// SIMATIC STEP 7 (V5.x) project PLC
// CPU: CPU 315-2 DP
// station: P_ADR_BUS
// station: Hardware
// station: SIMATIC 300(1)
// program: Programma S7(1)

// FB 2: know-how protected block, not included

// FB 3: know-how protected block, not included

// FB 4: know-how protected block, not included

// FB 6: know-how protected block, not included

// FC 1: know-how protected block, not included

FUNCTION FC 2 : VOID
VERSION : 0.1
BEGIN
// (block stored without names or comments; labels and parameter names are numbered)
NETWORK
TITLE =
      TAR1  LD 22;
NETWORK
TITLE =
      LAR1  P#L 2.0;
      L     B#16#10;
      T     LB [AR1,P#0.0];
      L     B#16#2;
      T     LB [AR1,P#1.0];
      L     #PARAM5;
      T     LW [AR1,P#2.0];
      L     #PARAM1;
      T     LW [AR1,P#4.0];
      L     P#DBX 0.0;
      L     #PARAM2;
      SLD   3;
      +D;
      T     LD [AR1,P#6.0];
NETWORK
TITLE =
      LAR1  P#L 12.0;
      L     B#16#10;
      T     LB [AR1,P#0.0];
      L     B#16#2;
      T     LB [AR1,P#1.0];
      L     #PARAM5;
      T     LW [AR1,P#2.0];
      L     #PARAM3;
      T     LW [AR1,P#4.0];
      L     P#DBX 0.0;
      L     #PARAM4;
      SLD   3;
      +D;
      T     LD [AR1,P#6.0];
NETWORK
TITLE =
      CALL  SFC 20 (
           $1                       := P#L 2.0,
           $2                       := P#L 0.0,
           $3                       := P#L 12.0);
NETWORK
TITLE =
      LAR1  LD 22;
END_FUNCTION

// FC 5: know-how protected block, not included

FUNCTION FC 8 : VOID
VERSION : 0.1
BEGIN
// (block stored without names or comments; labels and parameter names are numbered)
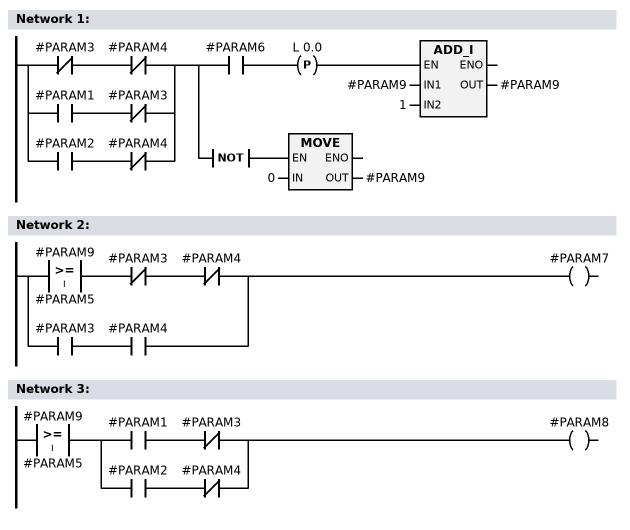
NETWORK
TITLE =
      AN    #PARAM3;
      AN    #PARAM4;
      O;
      A     #PARAM1;
      AN    #PARAM3;
      O;
      A     #PARAM2;
      AN    #PARAM4;
      =     L 1.0;
      A     L 1.0;
      A     #PARAM6;
      FP    L 0.0;
      JNB   M001;
      L     #PARAM9;
      L     1;
      +I;
      T     #PARAM9;
M001: NOP   0;
      A     L 1.0;
      NOT;
      JNB   M002;
      L     0;
      T     #PARAM9;
M002: NOP   0;
NETWORK
TITLE =
      A(;
      L     #PARAM9;
      L     #PARAM5;
      >=I;
      );
      AN    #PARAM3;
      AN    #PARAM4;
      O;
      A     #PARAM3;
      A     #PARAM4;
      =     #PARAM7;
NETWORK
TITLE =
      A(;
      L     #PARAM9;
      L     #PARAM5;
      >=I;
      );
      A(;
      A     #PARAM1;
      AN    #PARAM3;
      O;
      A     #PARAM2;
      AN    #PARAM4;
      );
      =     #PARAM8;
END_FUNCTION

// FC 20: know-how protected block, not included

// FC 21: know-how protected block, not included

// FC 22: know-how protected block, not included

// FC 23: know-how protected block, not included

FUNCTION FC 100 : VOID
VERSION : 0.1
BEGIN
// (block stored without names or comments; labels and parameter names are numbered)
NETWORK
TITLE =
      AN    DB30.DBX 7.0;
      =     DB30.DBX 6.0;
NETWORK
TITLE =
      AN    DB30.DBX 9.0;
      =     DB30.DBX 8.0;
NETWORK
TITLE =
      AN    DB30.DBX 7.1;
      =     DB30.DBX 6.1;
NETWORK
TITLE =
      AN    DB30.DBX 9.1;
      =     DB30.DBX 8.1;
NETWORK
TITLE =
      AN    DB30.DBX 21.1;
      =     DB30.DBX 21.1;
NETWORK
TITLE =
      AN    DB30.DBX 21.2;
      =     DB30.DBX 21.2;
NETWORK
TITLE =
NETWORK
TITLE =
      A     I 6.0;
      =     DB31.DBX 7.7;
NETWORK
TITLE =
      A     I 6.1;
      =     DB31.DBX 107.7;
NETWORK
TITLE =
      A     I 40.5;
      =     DB31.DBX 207.7;
NETWORK
TITLE =
NETWORK
TITLE =
      A     M 10.4;
      A(;
      L     DB30.DBW 34;
      L     18;
      <>I;
      );
      A(;
      L     DB30.DBW 34;
      L     28;
      <>I;
      );
      A(;
      O     I 102.5;
      O     DB30.DBX 509.0;
      );
      =     DB30.DBX 509.0;
NETWORK
TITLE =
      A     M 100.1;
      AN    Q 102.0;
      AN    Q 102.2;
      =     DB30.DBX 509.1;
NETWORK
TITLE =
      A     M 100.3;
      AN    Q 102.1;
      AN    Q 102.3;
      =     DB30.DBX 509.2;
NETWORK
TITLE =
      A     I 60.0;
      A     I 60.1;
      A     I 60.4;
      AN    DB100.DBX 110.0;
      =     DB30.DBX 509.3;
NETWORK
TITLE =
      A     I 60.0;
      A     I 60.1;
      AN    DB100.DBX 110.0;
      =     DB30.DBX 509.4;
NETWORK
TITLE =
      A     I 70.0;
      A     I 70.1;
      A     I 70.4;
      AN    DB100.DBX 110.1;
      =     DB30.DBX 509.5;
NETWORK
TITLE =
      A     I 70.0;
      A     I 70.1;
      AN    DB100.DBX 110.1;
      =     DB30.DBX 509.6;
NETWORK
TITLE =
      A     M 136.2;
      =     DB30.DBX 509.7;
NETWORK
TITLE =
      A     I 80.1;
      AN    DB100.DBX 110.2;
      =     DB30.DBX 511.0;
NETWORK
TITLE =
      A     DB100.DBX 110.6;
      =     DB30.DBX 511.1;
NETWORK
TITLE =
      A     I 90.1;
      AN    DB100.DBX 110.5;
      =     DB30.DBX 511.2;
NETWORK
TITLE =
      A     DB100.DBX 111.0;
      =     DB30.DBX 511.3;
NETWORK
TITLE =
      A     DB100.DBX 111.1;
      =     DB30.DBX 511.4;
NETWORK
TITLE =
      A     M 10.6;
      =     DB30.DBX 511.6;
NETWORK
TITLE =
      A     M 100.0;
      A     M 100.2;
      =     DB30.DBX 511.7;
END_FUNCTION

FUNCTION FC 101 : VOID
VERSION : 0.1
BEGIN
// (block stored without names or comments; labels and parameter names are numbered)
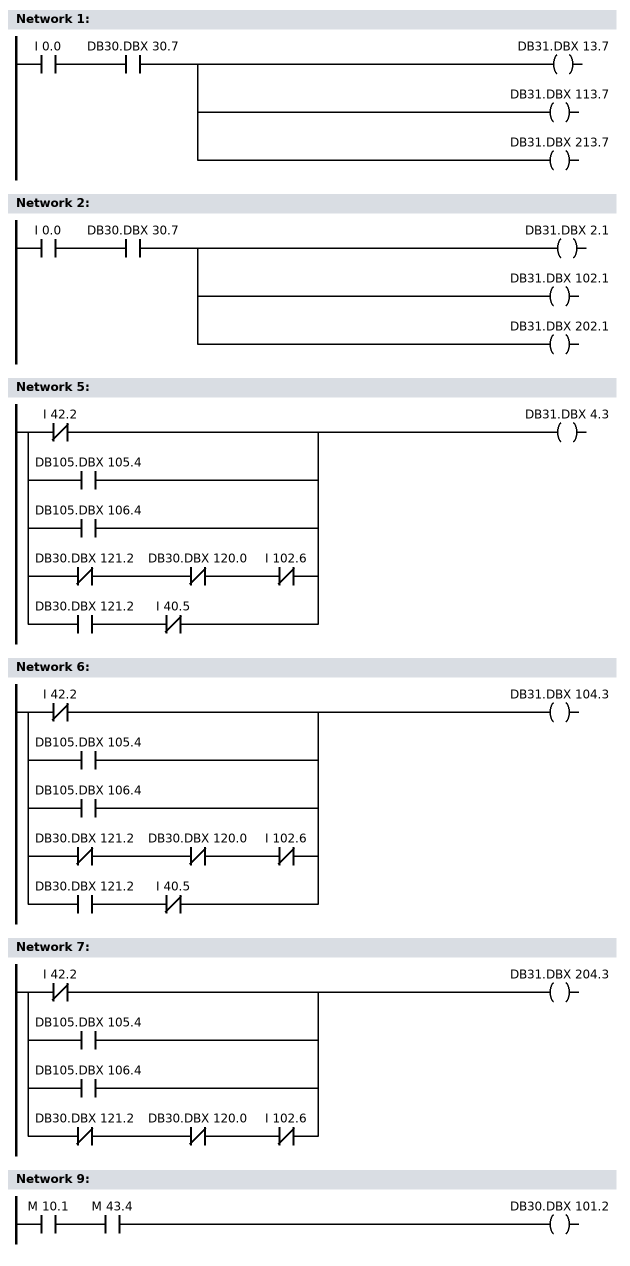
NETWORK
TITLE =
      A     I 0.0;
      A     DB30.DBX 30.7;
      =     DB31.DBX 13.7;
      =     DB31.DBX 113.7;
      =     DB31.DBX 213.7;
NETWORK
TITLE =
      A     I 0.0;
      A     DB30.DBX 30.7;
      =     DB31.DBX 2.1;
      =     DB31.DBX 102.1;
      =     DB31.DBX 202.1;
NETWORK
TITLE =
NETWORK
TITLE =
NETWORK
TITLE =
      ON    I 42.2;
      O     DB105.DBX 105.4;
      O     DB105.DBX 106.4;
      O;
      AN    DB30.DBX 121.2;
      AN    DB30.DBX 120.0;
      AN    I 102.6;
      O;
      A     DB30.DBX 121.2;
      AN    I 40.5;
      =     DB31.DBX 4.3;
NETWORK
TITLE =
      ON    I 42.2;
      O     DB105.DBX 105.4;
      O     DB105.DBX 106.4;
      O;
      AN    DB30.DBX 121.2;
      AN    DB30.DBX 120.0;
      AN    I 102.6;
      O;
      A     DB30.DBX 121.2;
      AN    I 40.5;
      =     DB31.DBX 104.3;
NETWORK
TITLE =
      ON    I 42.2;
      O     DB105.DBX 105.4;
      O     DB105.DBX 106.4;
      O;
      AN    DB30.DBX 121.2;
      AN    DB30.DBX 120.0;
      AN    I 102.6;
      =     DB31.DBX 204.3;
NETWORK
TITLE =
NETWORK
TITLE =
      A     M 10.1;
      A     M 43.4;
      =     DB30.DBX 101.2;
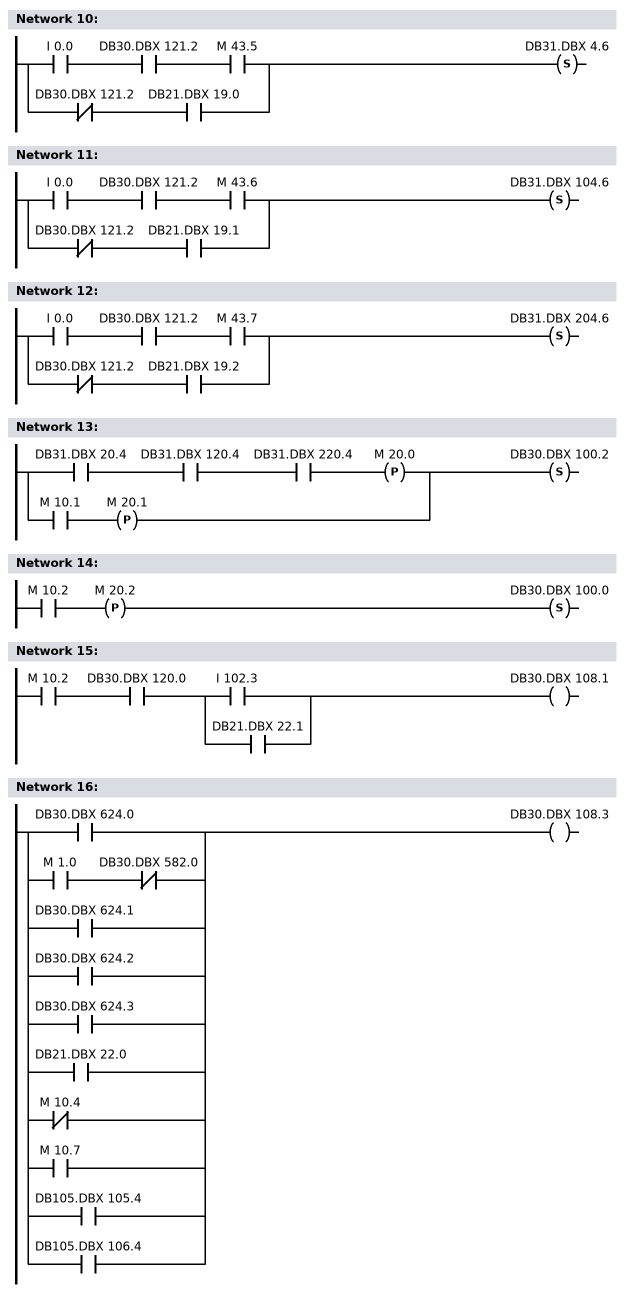
NETWORK
TITLE =
      A     I 0.0;
      A     DB30.DBX 121.2;
      A     M 43.5;
      O;
      AN    DB30.DBX 121.2;
      A     DB21.DBX 19.0;
      S     DB31.DBX 4.6;
NETWORK
TITLE =
      A     I 0.0;
      A     DB30.DBX 121.2;
      A     M 43.6;
      O;
      AN    DB30.DBX 121.2;
      A     DB21.DBX 19.1;
      S     DB31.DBX 104.6;
NETWORK
TITLE =
      A     I 0.0;
      A     DB30.DBX 121.2;
      A     M 43.7;
      O;
      AN    DB30.DBX 121.2;
      A     DB21.DBX 19.2;
      S     DB31.DBX 204.6;
NETWORK
TITLE =
      A     DB31.DBX 20.4;
      A     DB31.DBX 120.4;
      A     DB31.DBX 220.4;
      FP    M 20.0;
      O(;
      A     M 10.1;
      FP    M 20.1;
      );
      S     DB30.DBX 100.2;
NETWORK
TITLE =
      A     M 10.2;
      FP    M 20.2;
      S     DB30.DBX 100.0;
NETWORK
TITLE =
      A     M 10.2;
      A     DB30.DBX 120.0;
      A(;
      O     I 102.3;
      O     DB21.DBX 22.1;
      );
      =     DB30.DBX 108.1;
NETWORK
TITLE =
      O     DB30.DBX 624.0;
      O;
      A     M 1.0;
      AN    DB30.DBX 582.0;
      O     DB30.DBX 624.1;
      O     DB30.DBX 624.2;
      O     DB30.DBX 624.3;
      O     DB21.DBX 22.0;
      ON    M 10.4;
      O     M 10.7;
      O     DB105.DBX 105.4;
      O     DB105.DBX 106.4;
      =     DB30.DBX 108.3;
END_FUNCTION

FUNCTION FC 102 : VOID
VERSION : 0.1
BEGIN
// (block stored without names or comments; labels and parameter names are numbered)
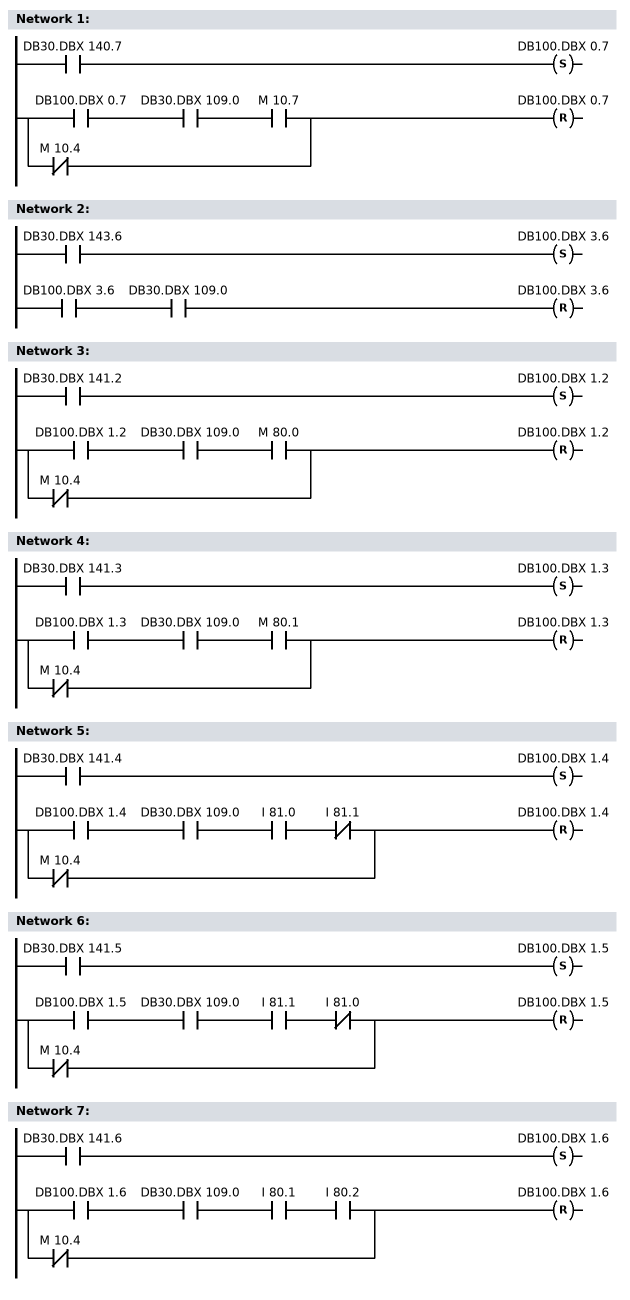
NETWORK
TITLE =
      A     DB30.DBX 140.7;
      S     DB100.DBX 0.7;
      A(;
      A     DB100.DBX 0.7;
      A     DB30.DBX 109.0;
      A     M 10.7;
      ON    M 10.4;
      );
      R     DB100.DBX 0.7;
      NOP   0;
NETWORK
TITLE =
      A     DB30.DBX 143.6;
      S     DB100.DBX 3.6;
      A     DB100.DBX 3.6;
      A     DB30.DBX 109.0;
      R     DB100.DBX 3.6;
      NOP   0;
NETWORK
TITLE =
      A     DB30.DBX 141.2;
      S     DB100.DBX 1.2;
      A(;
      A     DB100.DBX 1.2;
      A     DB30.DBX 109.0;
      A     M 80.0;
      ON    M 10.4;
      );
      R     DB100.DBX 1.2;
      NOP   0;
NETWORK
TITLE =
      A     DB30.DBX 141.3;
      S     DB100.DBX 1.3;
      A(;
      A     DB100.DBX 1.3;
      A     DB30.DBX 109.0;
      A     M 80.1;
      ON    M 10.4;
      );
      R     DB100.DBX 1.3;
      NOP   0;
NETWORK
TITLE =
      A     DB30.DBX 141.4;
      S     DB100.DBX 1.4;
      A(;
      A     DB100.DBX 1.4;
      A     DB30.DBX 109.0;
      A     I 81.0;
      AN    I 81.1;
      ON    M 10.4;
      );
      R     DB100.DBX 1.4;
      NOP   0;
NETWORK
TITLE =
      A     DB30.DBX 141.5;
      S     DB100.DBX 1.5;
      A(;
      A     DB100.DBX 1.5;
      A     DB30.DBX 109.0;
      A     I 81.1;
      AN    I 81.0;
      ON    M 10.4;
      );
      R     DB100.DBX 1.5;
      NOP   0;
NETWORK
TITLE =
      A     DB30.DBX 141.6;
      S     DB100.DBX 1.6;
      A(;
      A     DB100.DBX 1.6;
      A     DB30.DBX 109.0;
      A     I 80.1;
      A     I 80.2;
      ON    M 10.4;
      );
      R     DB100.DBX 1.6;
      NOP   0;
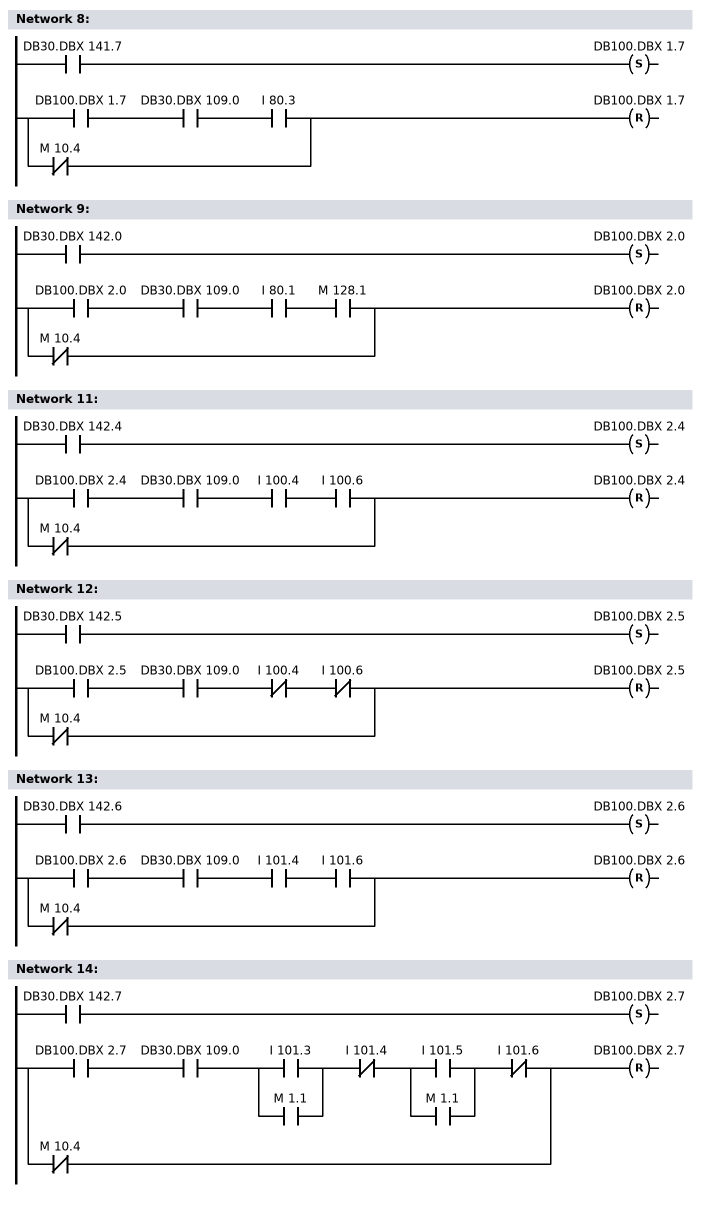
NETWORK
TITLE =
      A     DB30.DBX 141.7;
      S     DB100.DBX 1.7;
      A(;
      A     DB100.DBX 1.7;
      A     DB30.DBX 109.0;
      A     I 80.3;
      ON    M 10.4;
      );
      R     DB100.DBX 1.7;
      NOP   0;
NETWORK
TITLE =
      A     DB30.DBX 142.0;
      S     DB100.DBX 2.0;
      A(;
      A     DB100.DBX 2.0;
      A     DB30.DBX 109.0;
      A     I 80.1;
      A     M 128.1;
      ON    M 10.4;
      );
      R     DB100.DBX 2.0;
      NOP   0;
NETWORK
TITLE =
NETWORK
TITLE =
      A     DB30.DBX 142.4;
      S     DB100.DBX 2.4;
      A(;
      A     DB100.DBX 2.4;
      A     DB30.DBX 109.0;
      A     I 100.4;
      A     I 100.6;
      ON    M 10.4;
      );
      R     DB100.DBX 2.4;
      NOP   0;
NETWORK
TITLE =
      A     DB30.DBX 142.5;
      S     DB100.DBX 2.5;
      A(;
      A     DB100.DBX 2.5;
      A     DB30.DBX 109.0;
      AN    I 100.4;
      AN    I 100.6;
      ON    M 10.4;
      );
      R     DB100.DBX 2.5;
      NOP   0;
NETWORK
TITLE =
      A     DB30.DBX 142.6;
      S     DB100.DBX 2.6;
      A(;
      A     DB100.DBX 2.6;
      A     DB30.DBX 109.0;
      A     I 101.4;
      A     I 101.6;
      ON    M 10.4;
      );
      R     DB100.DBX 2.6;
      NOP   0;
NETWORK
TITLE =
      A     DB30.DBX 142.7;
      S     DB100.DBX 2.7;
      A(;
      A     DB100.DBX 2.7;
      A     DB30.DBX 109.0;
      A(;
      O     I 101.3;
      O     M 1.1;
      );
      AN    I 101.4;
      A(;
      O     I 101.5;
      O     M 1.1;
      );
      AN    I 101.6;
      ON    M 10.4;
      );
      R     DB100.DBX 2.7;
      NOP   0;
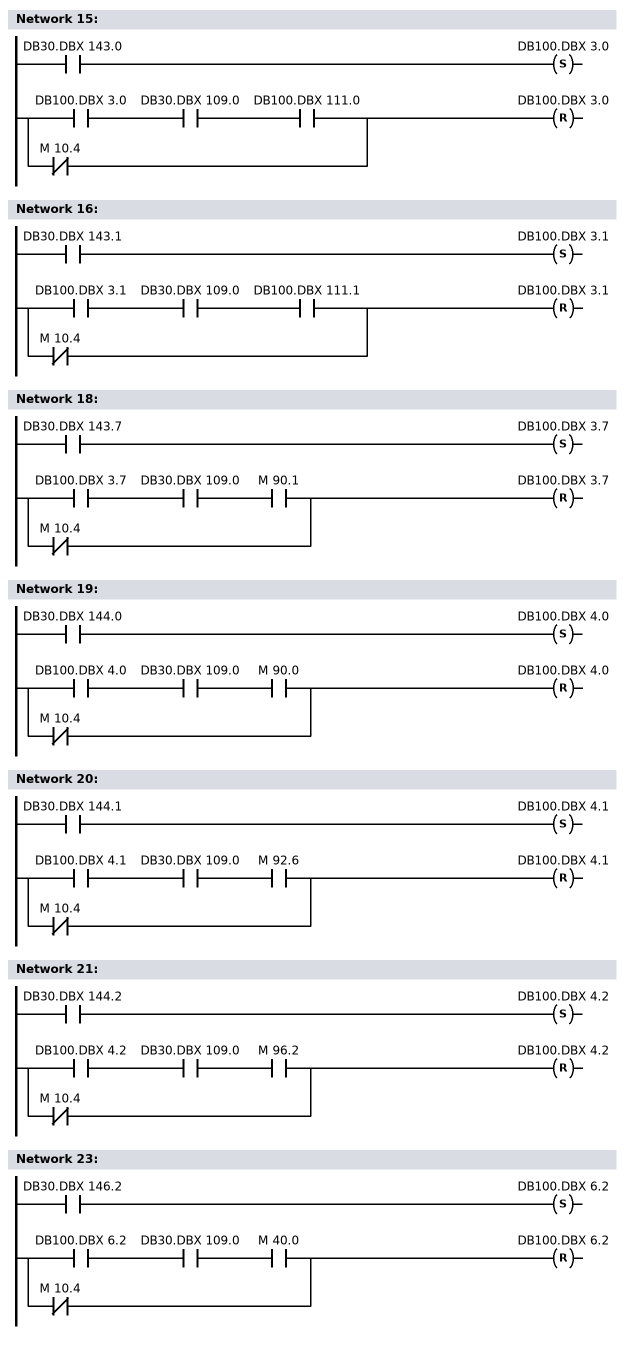
NETWORK
TITLE =
      A     DB30.DBX 143.0;
      S     DB100.DBX 3.0;
      A(;
      A     DB100.DBX 3.0;
      A     DB30.DBX 109.0;
      A     DB100.DBX 111.0;
      ON    M 10.4;
      );
      R     DB100.DBX 3.0;
      NOP   0;
NETWORK
TITLE =
      A     DB30.DBX 143.1;
      S     DB100.DBX 3.1;
      A(;
      A     DB100.DBX 3.1;
      A     DB30.DBX 109.0;
      A     DB100.DBX 111.1;
      ON    M 10.4;
      );
      R     DB100.DBX 3.1;
      NOP   0;
NETWORK
TITLE =
NETWORK
TITLE =
      A     DB30.DBX 143.7;
      S     DB100.DBX 3.7;
      A(;
      A     DB100.DBX 3.7;
      A     DB30.DBX 109.0;
      A     M 90.1;
      ON    M 10.4;
      );
      R     DB100.DBX 3.7;
      NOP   0;
NETWORK
TITLE =
      A     DB30.DBX 144.0;
      S     DB100.DBX 4.0;
      A(;
      A     DB100.DBX 4.0;
      A     DB30.DBX 109.0;
      A     M 90.0;
      ON    M 10.4;
      );
      R     DB100.DBX 4.0;
      NOP   0;
NETWORK
TITLE =
      A     DB30.DBX 144.1;
      S     DB100.DBX 4.1;
      A(;
      A     DB100.DBX 4.1;
      A     DB30.DBX 109.0;
      A     M 92.6;
      ON    M 10.4;
      );
      R     DB100.DBX 4.1;
      NOP   0;
NETWORK
TITLE =
      A     DB30.DBX 144.2;
      S     DB100.DBX 4.2;
      A(;
      A     DB100.DBX 4.2;
      A     DB30.DBX 109.0;
      A     M 96.2;
      ON    M 10.4;
      );
      R     DB100.DBX 4.2;
      NOP   0;
NETWORK
TITLE =
NETWORK
TITLE =
      A     DB30.DBX 146.2;
      S     DB100.DBX 6.2;
      A(;
      A     DB100.DBX 6.2;
      A     DB30.DBX 109.0;
      A     M 40.0;
      ON    M 10.4;
      );
      R     DB100.DBX 6.2;
      NOP   0;
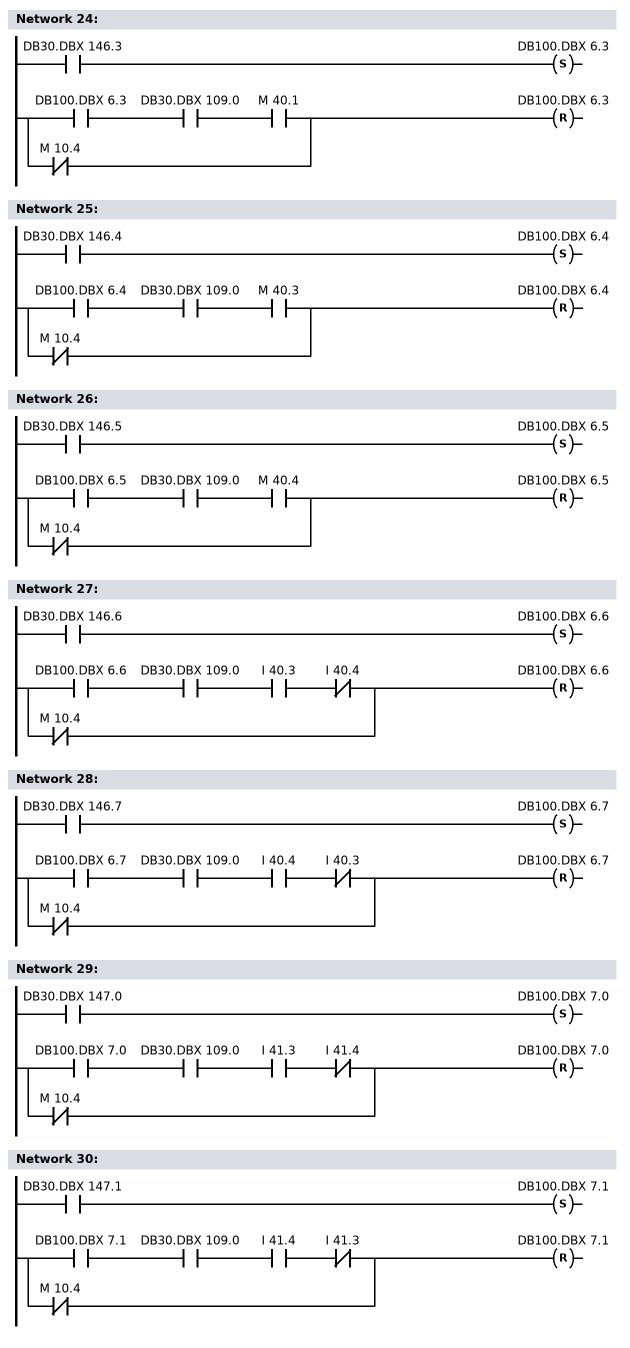
NETWORK
TITLE =
      A     DB30.DBX 146.3;
      S     DB100.DBX 6.3;
      A(;
      A     DB100.DBX 6.3;
      A     DB30.DBX 109.0;
      A     M 40.1;
      ON    M 10.4;
      );
      R     DB100.DBX 6.3;
      NOP   0;
NETWORK
TITLE =
      A     DB30.DBX 146.4;
      S     DB100.DBX 6.4;
      A(;
      A     DB100.DBX 6.4;
      A     DB30.DBX 109.0;
      A     M 40.3;
      ON    M 10.4;
      );
      R     DB100.DBX 6.4;
      NOP   0;
NETWORK
TITLE =
      A     DB30.DBX 146.5;
      S     DB100.DBX 6.5;
      A(;
      A     DB100.DBX 6.5;
      A     DB30.DBX 109.0;
      A     M 40.4;
      ON    M 10.4;
      );
      R     DB100.DBX 6.5;
      NOP   0;
NETWORK
TITLE =
      A     DB30.DBX 146.6;
      S     DB100.DBX 6.6;
      A(;
      A     DB100.DBX 6.6;
      A     DB30.DBX 109.0;
      A     I 40.3;
      AN    I 40.4;
      ON    M 10.4;
      );
      R     DB100.DBX 6.6;
      NOP   0;
NETWORK
TITLE =
      A     DB30.DBX 146.7;
      S     DB100.DBX 6.7;
      A(;
      A     DB100.DBX 6.7;
      A     DB30.DBX 109.0;
      A     I 40.4;
      AN    I 40.3;
      ON    M 10.4;
      );
      R     DB100.DBX 6.7;
      NOP   0;
NETWORK
TITLE =
      A     DB30.DBX 147.0;
      S     DB100.DBX 7.0;
      A(;
      A     DB100.DBX 7.0;
      A     DB30.DBX 109.0;
      A     I 41.3;
      AN    I 41.4;
      ON    M 10.4;
      );
      R     DB100.DBX 7.0;
      NOP   0;
NETWORK
TITLE =
      A     DB30.DBX 147.1;
      S     DB100.DBX 7.1;
      A(;
      A     DB100.DBX 7.1;
      A     DB30.DBX 109.0;
      A     I 41.4;
      AN    I 41.3;
      ON    M 10.4;
      );
      R     DB100.DBX 7.1;
      NOP   0;
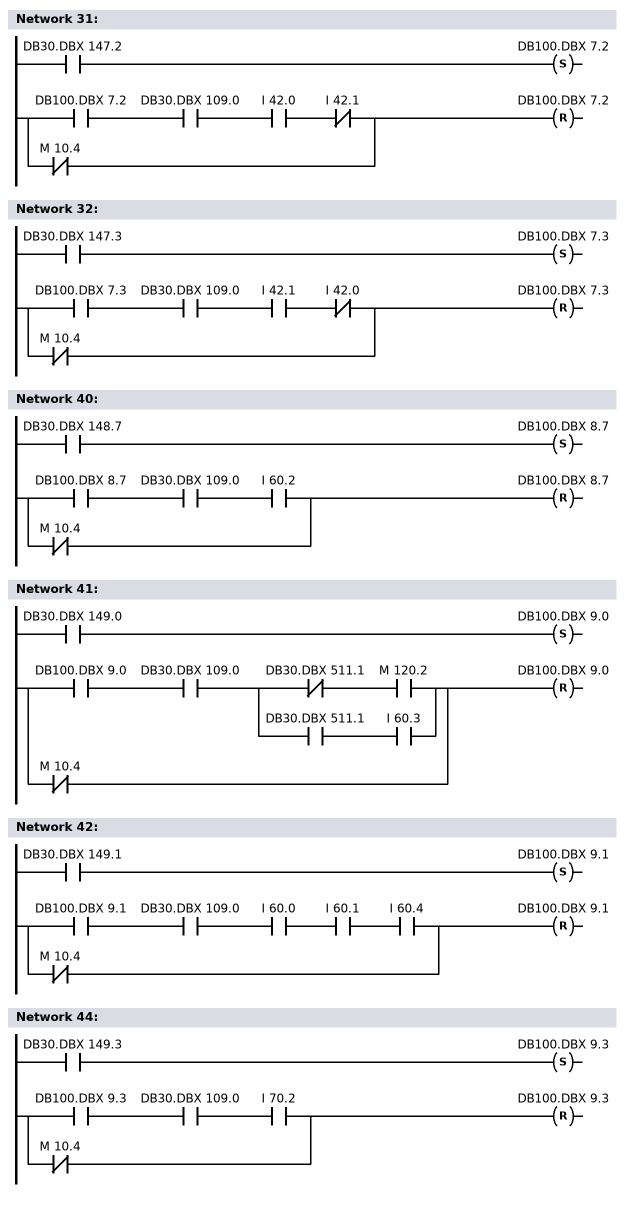
NETWORK
TITLE =
      A     DB30.DBX 147.2;
      S     DB100.DBX 7.2;
      A(;
      A     DB100.DBX 7.2;
      A     DB30.DBX 109.0;
      A     I 42.0;
      AN    I 42.1;
      ON    M 10.4;
      );
      R     DB100.DBX 7.2;
      NOP   0;
NETWORK
TITLE =
      A     DB30.DBX 147.3;
      S     DB100.DBX 7.3;
      A(;
      A     DB100.DBX 7.3;
      A     DB30.DBX 109.0;
      A     I 42.1;
      AN    I 42.0;
      ON    M 10.4;
      );
      R     DB100.DBX 7.3;
      NOP   0;
NETWORK
TITLE =
      A(;
      A     DB30.DBX 147.4;
      S     DB100.DBX 7.4;
      A(;
      A     DB100.DBX 7.4;
      A     DB30.DBX 109.0;
      A     M 132.0;
      ON    M 10.4;
      );
      R     DB100.DBX 7.4;
      A     DB100.DBX 7.4;
      );
      S     M 132.0;
      A     M 132.0;
      AN    DB100.DBX 7.4;
      A     I 40.3;
      AN    I 40.4;
      AN    I 41.3;
      A     I 41.4;
      AN    I 42.0;
      A     I 42.1;
      R     M 132.0;
      NOP   0;
NETWORK
TITLE =
      A(;
      A     DB30.DBX 147.5;
      S     DB100.DBX 7.5;
      A(;
      A     DB100.DBX 7.5;
      A     DB30.DBX 109.0;
      A     M 132.1;
      ON    M 10.4;
      );
      R     DB100.DBX 7.5;
      A     DB100.DBX 7.5;
      );
      S     M 132.1;
      A     M 132.1;
      AN    DB100.DBX 7.5;
      AN    I 40.3;
      A     I 40.4;
      A     I 41.3;
      AN    I 41.4;
      AN    I 42.0;
      A     I 42.1;
      R     M 132.1;
      NOP   0;
NETWORK
TITLE =
      A(;
      A     DB30.DBX 147.6;
      S     DB100.DBX 7.6;
      A(;
      A     DB100.DBX 7.6;
      A     DB30.DBX 109.0;
      A     M 132.2;
      ON    M 10.4;
      );
      R     DB100.DBX 7.6;
      A     DB100.DBX 7.6;
      );
      S     M 132.2;
      A     M 132.2;
      AN    DB100.DBX 7.6;
      A     I 40.3;
      AN    I 40.4;
      AN    I 41.3;
      A     I 41.4;
      A     I 42.0;
      AN    I 42.1;
      R     M 132.2;
      NOP   0;
NETWORK
TITLE =
      A(;
      A     DB30.DBX 147.7;
      S     DB100.DBX 7.7;
      A(;
      A     DB100.DBX 7.7;
      A     DB30.DBX 109.0;
      A     M 132.3;
      ON    M 10.4;
      );
      R     DB100.DBX 7.7;
      A     DB100.DBX 7.7;
      );
      S     M 132.3;
      A     M 132.3;
      AN    DB100.DBX 7.7;
      AN    I 40.3;
      A     I 40.4;
      A     I 41.3;
      AN    I 41.4;
      A     I 42.0;
      AN    I 42.1;
      R     M 132.3;
      NOP   0;
NETWORK
TITLE =
      A(;
      A     DB30.DBX 148.0;
      S     DB100.DBX 8.0;
      A(;
      A     DB100.DBX 8.0;
      A     DB30.DBX 109.0;
      A     M 132.4;
      ON    M 10.4;
      );
      R     DB100.DBX 8.0;
      A     DB100.DBX 8.0;
      );
      S     M 132.4;
      A     M 132.4;
      AN    DB100.DBX 8.0;
      AN    I 40.3;
      A     I 40.4;
      AN    I 41.3;
      A     I 41.4;
      A     I 42.0;
      AN    I 42.1;
      R     M 132.4;
      NOP   0;
NETWORK
TITLE =
      A(;
      A     DB30.DBX 148.1;
      S     DB100.DBX 8.1;
      A(;
      A     DB100.DBX 8.1;
      A     DB30.DBX 109.0;
      A     M 132.5;
      ON    M 10.4;
      );
      R     DB100.DBX 8.1;
      A     DB100.DBX 8.1;
      );
      S     M 132.5;
      A     M 132.5;
      AN    DB100.DBX 8.1;
      AN    I 40.3;
      A     I 40.4;
      AN    I 41.3;
      A     I 41.4;
      AN    I 42.0;
      A     I 42.1;
      R     M 132.5;
      NOP   0;
NETWORK
TITLE =
NETWORK
TITLE =
      A     DB30.DBX 148.7;
      S     DB100.DBX 8.7;
      A(;
      A     DB100.DBX 8.7;
      A     DB30.DBX 109.0;
      A     I 60.2;
      ON    M 10.4;
      );
      R     DB100.DBX 8.7;
      NOP   0;
NETWORK
TITLE =
      A     DB30.DBX 149.0;
      S     DB100.DBX 9.0;
      A(;
      A     DB100.DBX 9.0;
      A     DB30.DBX 109.0;
      A(;
      AN    DB30.DBX 511.1;
      A     M 120.2;
      O;
      A     DB30.DBX 511.1;
      A     I 60.3;
      );
      ON    M 10.4;
      );
      R     DB100.DBX 9.0;
      NOP   0;
NETWORK
TITLE =
      A     DB30.DBX 149.1;
      S     DB100.DBX 9.1;
      A(;
      A     DB100.DBX 9.1;
      A     DB30.DBX 109.0;
      A     I 60.0;
      A     I 60.1;
      A     I 60.4;
      ON    M 10.4;
      );
      R     DB100.DBX 9.1;
      NOP   0;
NETWORK
TITLE =
NETWORK
TITLE =
      A     DB30.DBX 149.3;
      S     DB100.DBX 9.3;
      A(;
      A     DB100.DBX 9.3;
      A     DB30.DBX 109.0;
      A     I 70.2;
      ON    M 10.4;
      );
      R     DB100.DBX 9.3;
      NOP   0;
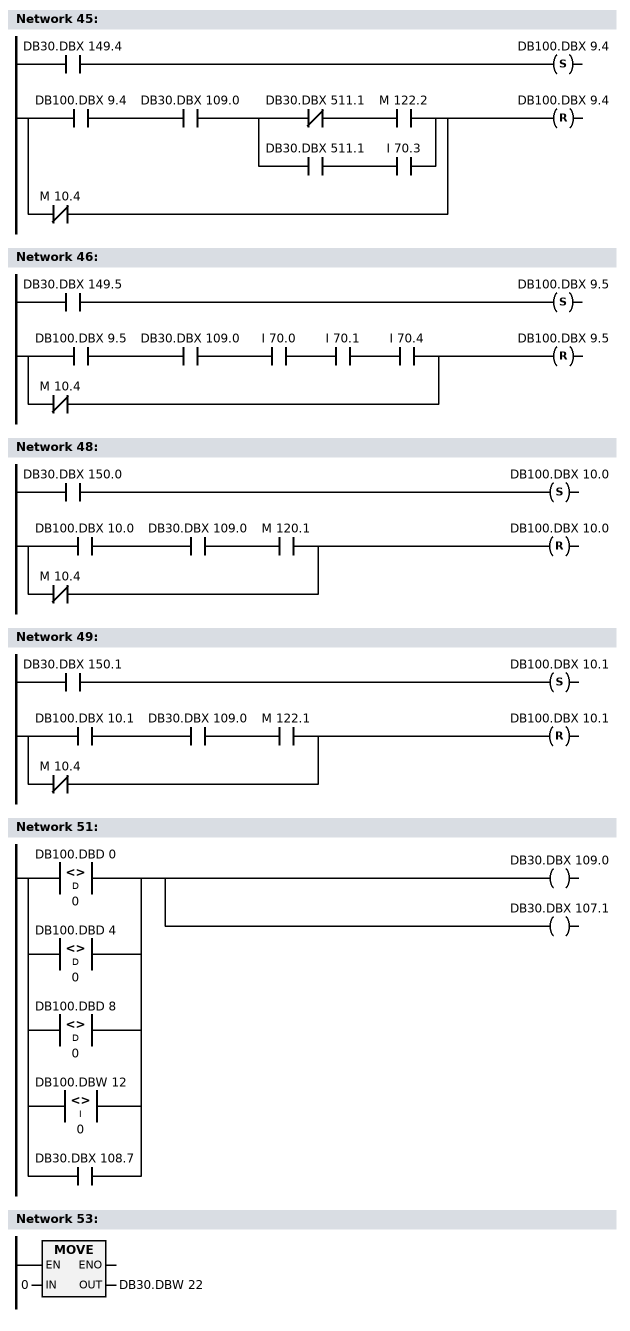
NETWORK
TITLE =
      A     DB30.DBX 149.4;
      S     DB100.DBX 9.4;
      A(;
      A     DB100.DBX 9.4;
      A     DB30.DBX 109.0;
      A(;
      AN    DB30.DBX 511.1;
      A     M 122.2;
      O;
      A     DB30.DBX 511.1;
      A     I 70.3;
      );
      ON    M 10.4;
      );
      R     DB100.DBX 9.4;
      NOP   0;
NETWORK
TITLE =
      A     DB30.DBX 149.5;
      S     DB100.DBX 9.5;
      A(;
      A     DB100.DBX 9.5;
      A     DB30.DBX 109.0;
      A     I 70.0;
      A     I 70.1;
      A     I 70.4;
      ON    M 10.4;
      );
      R     DB100.DBX 9.5;
      NOP   0;
NETWORK
TITLE =
NETWORK
TITLE =
      A     DB30.DBX 150.0;
      S     DB100.DBX 10.0;
      A(;
      A     DB100.DBX 10.0;
      A     DB30.DBX 109.0;
      A     M 120.1;
      ON    M 10.4;
      );
      R     DB100.DBX 10.0;
      NOP   0;
NETWORK
TITLE =
      A     DB30.DBX 150.1;
      S     DB100.DBX 10.1;
      A(;
      A     DB100.DBX 10.1;
      A     DB30.DBX 109.0;
      A     M 122.1;
      ON    M 10.4;
      );
      R     DB100.DBX 10.1;
      NOP   0;
NETWORK
TITLE =
NETWORK
TITLE =
      O(;
      L     DB100.DBD 0;
      L     0;
      <>D;
      );
      O(;
      L     DB100.DBD 4;
      L     0;
      <>D;
      );
      O(;
      L     DB100.DBD 8;
      L     0;
      <>D;
      );
      O(;
      L     DB100.DBW 12;
      L     0;
      <>I;
      );
      O     DB30.DBX 108.7;
      =     DB30.DBX 109.0;
      =     DB30.DBX 107.1;
NETWORK
TITLE =
NETWORK
TITLE =
      L     0;
      T     DB30.DBW 22;
      NOP   0;
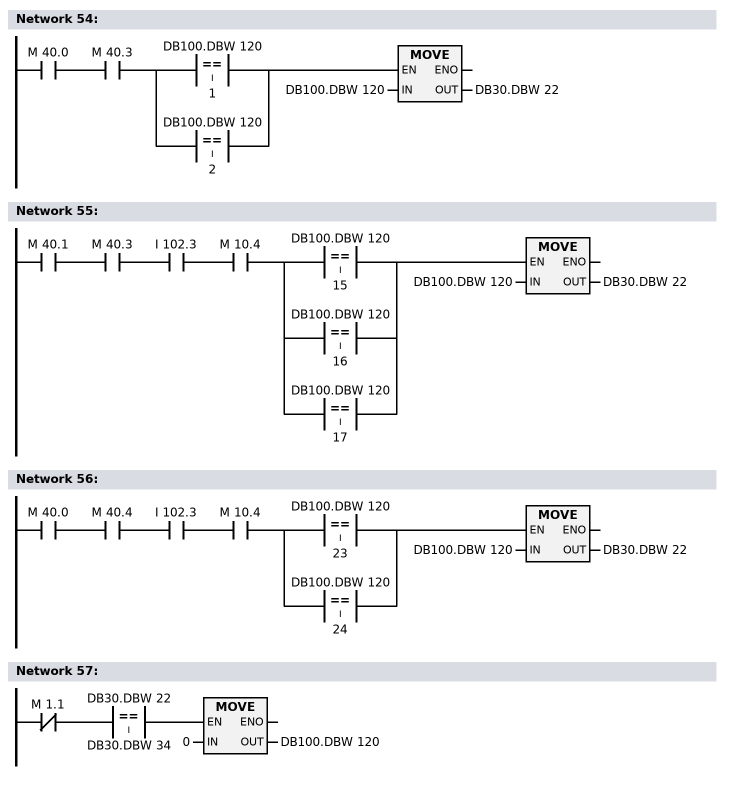
NETWORK
TITLE =
      A     M 40.0;
      A     M 40.3;
      A(;
      O(;
      L     DB100.DBW 120;
      L     1;
      ==I;
      );
      O(;
      L     DB100.DBW 120;
      L     2;
      ==I;
      );
      );
      JNB   M001;
      L     DB100.DBW 120;
      T     DB30.DBW 22;
M001: NOP   0;
NETWORK
TITLE =
      A     M 40.1;
      A     M 40.3;
      A     I 102.3;
      A     M 10.4;
      A(;
      O(;
      L     DB100.DBW 120;
      L     15;
      ==I;
      );
      O(;
      L     DB100.DBW 120;
      L     16;
      ==I;
      );
      O(;
      L     DB100.DBW 120;
      L     17;
      ==I;
      );
      );
      JNB   M002;
      L     DB100.DBW 120;
      T     DB30.DBW 22;
M002: NOP   0;
NETWORK
TITLE =
      A     M 40.0;
      A     M 40.4;
      A     I 102.3;
      A     M 10.4;
      A(;
      O(;
      L     DB100.DBW 120;
      L     23;
      ==I;
      );
      O(;
      L     DB100.DBW 120;
      L     24;
      ==I;
      );
      );
      JNB   M003;
      L     DB100.DBW 120;
      T     DB30.DBW 22;
M003: NOP   0;
NETWORK
TITLE =
      AN    M 1.1;
      A(;
      L     DB30.DBW 22;
      L     DB30.DBW 34;
      ==I;
      );
      JNB   M004;
      L     0;
      T     DB100.DBW 120;
M004: NOP   0;
END_FUNCTION

FUNCTION FC 104 : VOID
AUTHOR : AuD_MCE8
FAMILY : FM357_2
NAME : EXAMPLE5
VERSION : 1.0
BEGIN
// (block stored without names or comments; labels and parameter names are numbered)
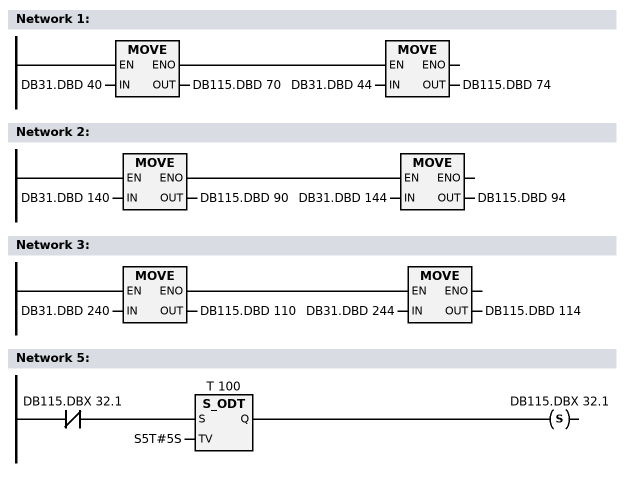
NETWORK
TITLE =
      A(;
      L     DB31.DBD 40;
      T     DB115.DBD 70;
      SET;
      SAVE;
      CLR;
      A     BR;
      );
      JNB   M001;
      L     DB31.DBD 44;
      T     DB115.DBD 74;
M001: NOP   0;
NETWORK
TITLE =
      A(;
      L     DB31.DBD 140;
      T     DB115.DBD 90;
      SET;
      SAVE;
      CLR;
      A     BR;
      );
      JNB   M002;
      L     DB31.DBD 144;
      T     DB115.DBD 94;
M002: NOP   0;
NETWORK
TITLE =
      A(;
      L     DB31.DBD 240;
      T     DB115.DBD 110;
      SET;
      SAVE;
      CLR;
      A     BR;
      );
      JNB   M003;
      L     DB31.DBD 244;
      T     DB115.DBD 114;
M003: NOP   0;
NETWORK
TITLE =
NETWORK
TITLE =
      AN    DB115.DBX 32.1;
      L     S5T#5S;
      SD    T 100;
      NOP   0;
      NOP   0;
      NOP   0;
      A     T 100;
      S     DB115.DBX 32.1;
NETWORK
TITLE =
      A     DB115.DBX 33.3;
      R     DB115.DBX 33.3;
      R     DB115.DBX 32.3;
      JC    M004;
      A     DB115.DBX 32.0;
      FP    DB115.DBX 33.5;
      S     DB115.DBX 32.3;
      O     DB115.DBX 32.7;
      O(;
      A     DB115.DBX 32.5;
      A     DB115.DBX 33.1;
      );
      R     DB115.DBX 32.3;
      R     DB115.DBX 32.0;
M004: CALL  FB 3 , DB 107 (
           DIX 0.0                  := DB115.DBX 32.3,
           DIW 2                    := 3,
           DIW 4                    := W#16#1002,
           DIW 6                    := 10,
           DIW 8                    := 121,
           DID 10                   := P#DBX 30.0,
           DIB 14                   := B#16#1,
           DIW 18                   := 1,
           DIW 132                  := 30,
           DIX 134.0                := DB115.DBX 33.1,
           DIX 134.1                := DB115.DBX 32.7,
           DIW 136                  := LW 0,
           DIW 138                  := W#16#1008,
           DIW 140                  := 1,
           DIW 142                  := 115,
           DID 144                  := P#DBX 0.0);
      L     B#16#0;
      A     DB115.DBX 33.1;
      JCN   M005;
      L     LW 0;
M005: T     DB115.DBW 30;
      A     DB115.DBX 33.2;
      R     DB115.DBX 33.2;
      R     DB115.DBX 32.2;
      JC    M006;
      A     DB115.DBX 32.1;
      FP    DB115.DBX 33.4;
      S     DB115.DBX 32.2;
      A     DB115.DBX 32.6;
      O(;
      A     DB115.DBX 32.4;
      A     DB115.DBX 33.0;
      );
      R     DB115.DBX 32.2;
      R     DB115.DBX 32.1;
M006: CALL  FB 2 , DB 106 (
           DIX 0.0                  := DB115.DBX 32.2,
           DIW 2                    := 8,
           DIW 4                    := W#16#1002,
           DIW 6                    := 10,
           DIW 8                    := 121,
           DID 10                   := P#DBX 30.0,
           DIB 14                   := B#16#1,
           DIW 18                   := 1,
           DIW 20                   := W#16#1002,
           DIW 22                   := 10,
           DIW 24                   := 121,
           DID 26                   := P#DBX 30.0,
           DIB 30                   := B#16#1,
           DIW 34                   := 2,
           DIW 36                   := W#16#1002,
           DIW 38                   := 10,
           DIW 40                   := 121,
           DID 42                   := P#DBX 30.0,
           DIB 46                   := B#16#1,
           DIW 50                   := 3,
           DIW 52                   := W#16#1002,
           DIW 54                   := 10,
           DIW 56                   := 121,
           DID 58                   := P#DBX 30.0,
           DIB 62                   := B#16#1,
           DIW 66                   := 4,
           DIW 68                   := W#16#1002,
           DIW 70                   := 10,
           DIW 72                   := 121,
           DID 74                   := P#DBX 30.0,
           DIB 78                   := B#16#1,
           DIW 82                   := 5,
           DIW 84                   := W#16#1002,
           DIW 86                   := 10,
           DIW 88                   := 121,
           DID 90                   := P#DBX 30.0,
           DIB 94                   := B#16#1,
           DIW 98                   := 6,
           DIW 100                  := W#16#1002,
           DIW 102                  := 10,
           DIW 104                  := 121,
           DID 106                  := P#DBX 30.0,
           DIB 110                  := B#16#1,
           DIW 114                  := 7,
           DIW 116                  := W#16#1002,
           DIW 118                  := 10,
           DIW 120                  := 121,
           DID 122                  := P#DBX 30.0,
           DIB 126                  := B#16#1,
           DIW 130                  := 8,
           DIW 132                  := 30,
           DIX 134.0                := DB115.DBX 33.0,
           DIX 134.1                := DB115.DBX 32.6,
           DIW 136                  := LW 0,
           DIW 138                  := W#16#1008,
           DIW 140                  := 1,
           DIW 142                  := 115,
           DID 144                  := P#DBX 34.0,
           DIW 148                  := W#16#1008,
           DIW 150                  := 1,
           DIW 152                  := 115,
           DID 154                  := P#DBX 38.0,
           DIW 158                  := W#16#1008,
           DIW 160                  := 1,
           DIW 162                  := 115,
           DID 164                  := P#DBX 42.0,
           DIW 168                  := W#16#1008,
           DIW 170                  := 1,
           DIW 172                  := 115,
           DID 174                  := P#DBX 46.0,
           DIW 178                  := W#16#1008,
           DIW 180                  := 1,
           DIW 182                  := 115,
           DID 184                  := P#DBX 50.0,
           DIW 188                  := W#16#1008,
           DIW 190                  := 1,
           DIW 192                  := 115,
           DID 194                  := P#DBX 54.0,
           DIW 198                  := W#16#1008,
           DIW 200                  := 1,
           DIW 202                  := 115,
           DID 204                  := P#DBX 58.0,
           DIW 208                  := W#16#1008,
           DIW 210                  := 1,
           DIW 212                  := 115,
           DID 214                  := P#DBX 62.0);
      L     B#16#0;
      A     DB115.DBX 33.0;
      JCN   M007;
      L     LW 0;
M007: T     DB115.DBW 28;
      BE;
END_FUNCTION

FUNCTION FC 110 : VOID
VERSION : 0.1
BEGIN
// (block stored without names or comments; labels and parameter names are numbered)
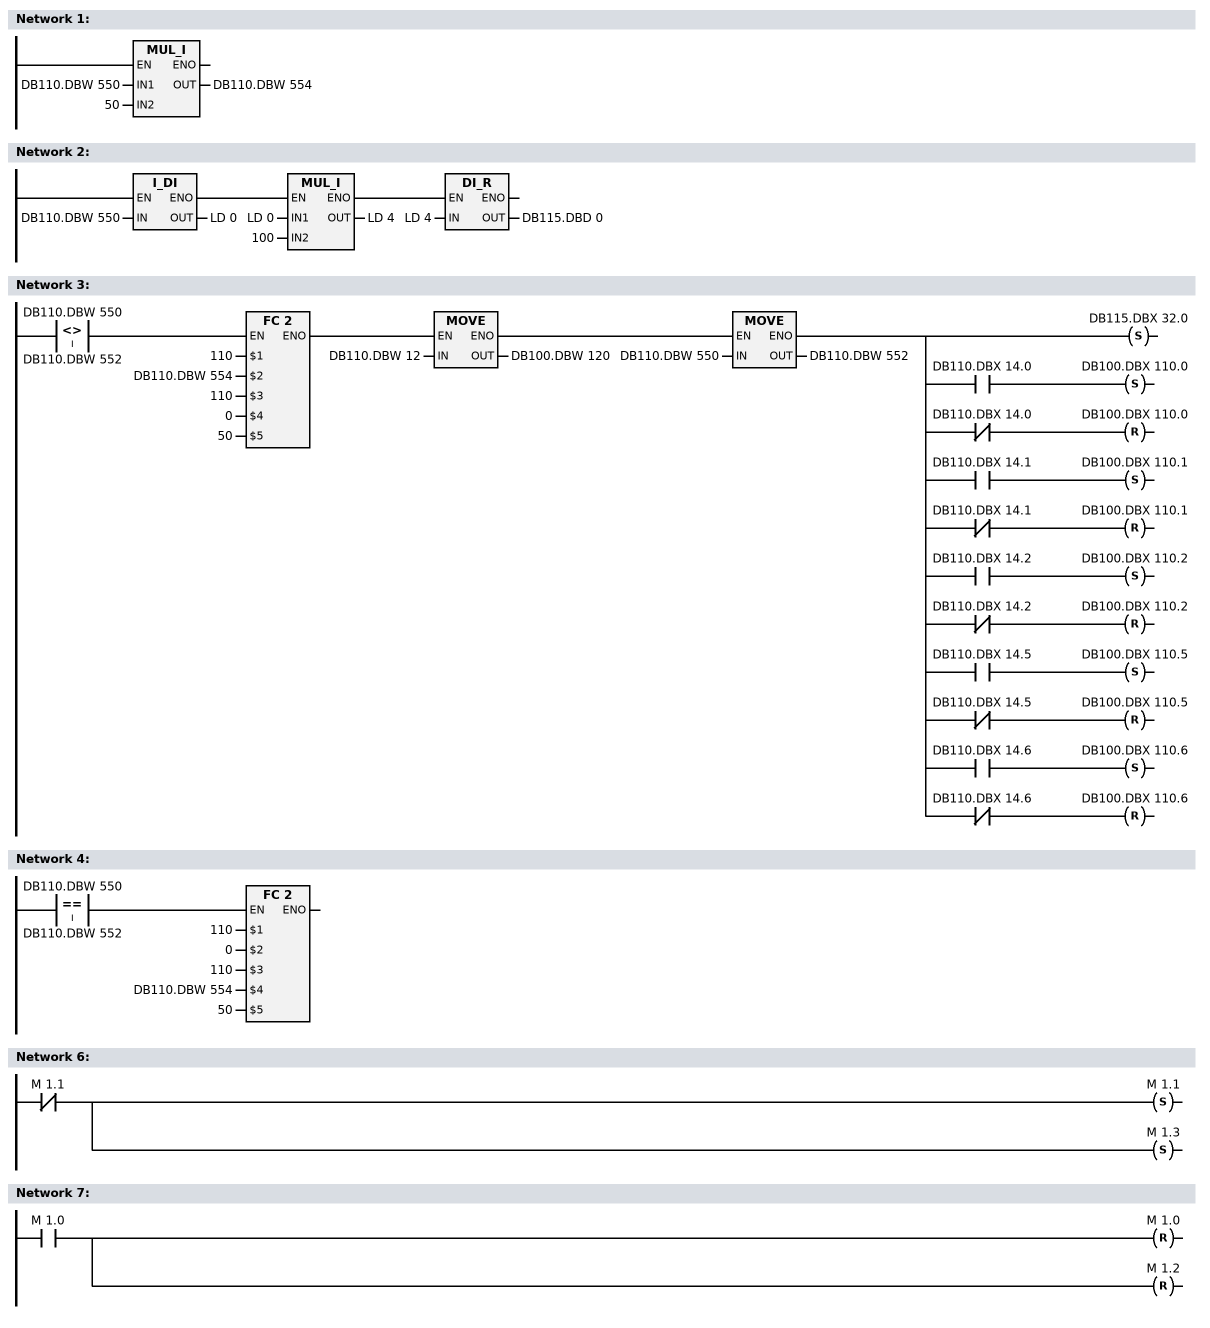
NETWORK
TITLE =
      L     DB110.DBW 550;
      L     50;
      *I;
      T     DB110.DBW 554;
      NOP   0;
NETWORK
TITLE =
      A(;
      A(;
      L     DB110.DBW 550;
      ITD;
      T     LD 0;
      SET;
      SAVE;
      CLR;
      A     BR;
      );
      JNB   M001;
      L     LD 0;
      L     100;
      *I;
      T     LD 4;
      AN    OV;
      SAVE;
      CLR;
M001: A     BR;
      );
      JNB   M002;
      L     LD 4;
      DTR;
      T     DB115.DBD 0;
M002: NOP   0;
NETWORK
TITLE =
      A(;
      A(;
      A(;
      L     DB110.DBW 550;
      L     DB110.DBW 552;
      <>I;
      );
      JNB   M003;
      CALL  FC 2 (
           $1                       := 110,
           $2                       := DB110.DBW 554,
           $3                       := 110,
           $4                       := 0,
           $5                       := 50);
M003: A     BR;
      );
      JNB   M004;
      L     DB110.DBW 12;
      T     DB100.DBW 120;
      SET;
      SAVE;
      CLR;
M004: A     BR;
      );
      JNB   M005;
      L     DB110.DBW 550;
      T     DB110.DBW 552;
      SET;
      SAVE;
      CLR;
M005: A     BR;
      =     L 8.0;
      A     L 8.0;
      BLD   102;
      S     DB115.DBX 32.0;
      A     L 8.0;
      A     DB110.DBX 14.0;
      S     DB100.DBX 110.0;
      A     L 8.0;
      AN    DB110.DBX 14.0;
      R     DB100.DBX 110.0;
      A     L 8.0;
      A     DB110.DBX 14.1;
      S     DB100.DBX 110.1;
      A     L 8.0;
      AN    DB110.DBX 14.1;
      R     DB100.DBX 110.1;
      A     L 8.0;
      A     DB110.DBX 14.2;
      S     DB100.DBX 110.2;
      A     L 8.0;
      AN    DB110.DBX 14.2;
      R     DB100.DBX 110.2;
      A     L 8.0;
      A     DB110.DBX 14.5;
      S     DB100.DBX 110.5;
      A     L 8.0;
      AN    DB110.DBX 14.5;
      R     DB100.DBX 110.5;
      A     L 8.0;
      A     DB110.DBX 14.6;
      S     DB100.DBX 110.6;
      A     L 8.0;
      AN    DB110.DBX 14.6;
      R     DB100.DBX 110.6;
NETWORK
TITLE =
      A(;
      L     DB110.DBW 550;
      L     DB110.DBW 552;
      ==I;
      );
      JNB   M006;
      CALL  FC 2 (
           $1                       := 110,
           $2                       := 0,
           $3                       := 110,
           $4                       := DB110.DBW 554,
           $5                       := 50);
M006: NOP   0;
NETWORK
TITLE =
NETWORK
TITLE =
      AN    M 1.1;
      S     M 1.1;
      S     M 1.3;
NETWORK
TITLE =
      A     M 1.0;
      R     M 1.0;
      R     M 1.2;
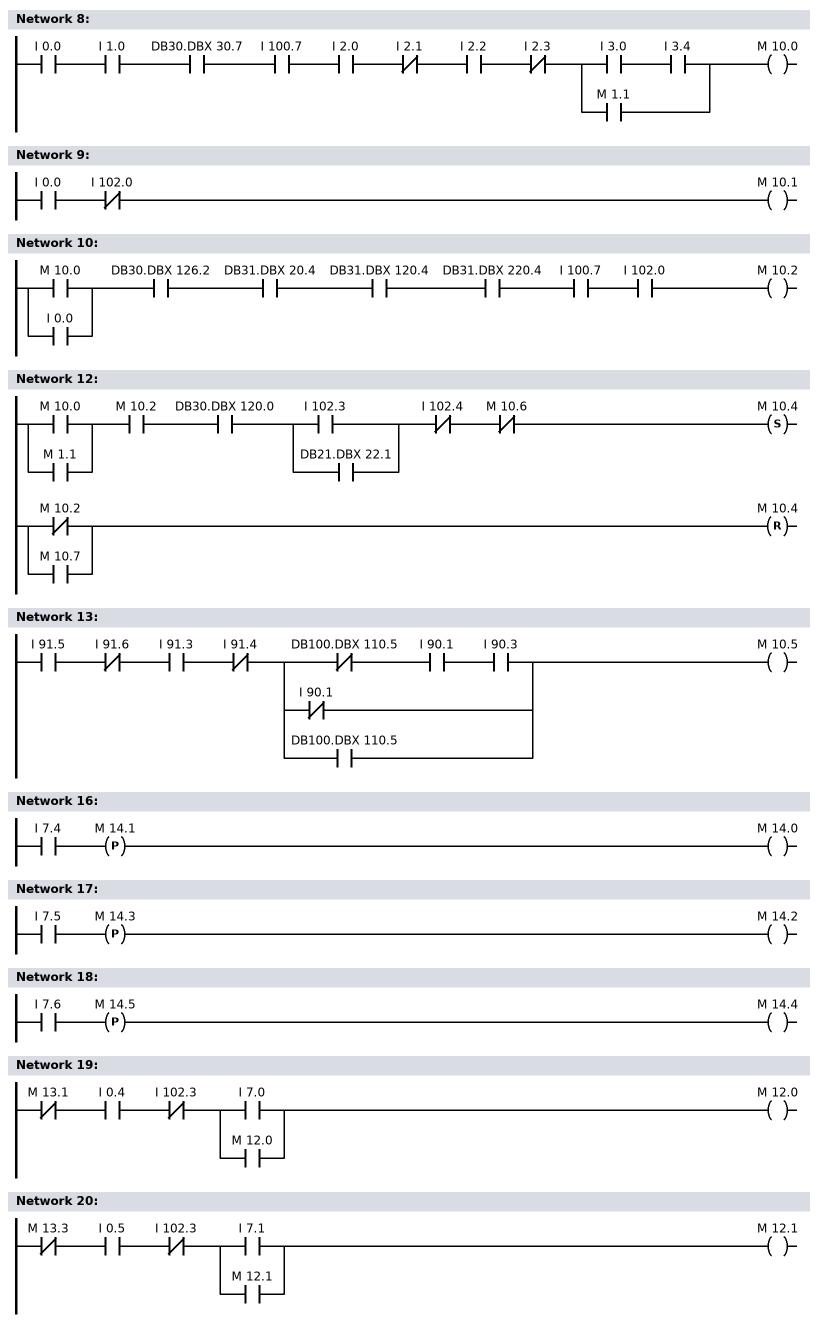
NETWORK
TITLE =
      A     I 0.0;
      A     I 1.0;
      A     DB30.DBX 30.7;
      A     I 100.7;
      A     I 2.0;
      AN    I 2.1;
      A     I 2.2;
      AN    I 2.3;
      A(;
      A     I 3.0;
      A     I 3.4;
      O     M 1.1;
      );
      =     M 10.0;
NETWORK
TITLE =
      A     I 0.0;
      AN    I 102.0;
      =     M 10.1;
NETWORK
TITLE =
      A(;
      O     M 10.0;
      O     I 0.0;
      );
      A     DB30.DBX 126.2;
      A     DB31.DBX 20.4;
      A     DB31.DBX 120.4;
      A     DB31.DBX 220.4;
      A     I 100.7;
      A     I 102.0;
      =     M 10.2;
NETWORK
TITLE =
NETWORK
TITLE =
      A(;
      O     M 10.0;
      O     M 1.1;
      );
      A     M 10.2;
      A     DB30.DBX 120.0;
      A(;
      O     I 102.3;
      O     DB21.DBX 22.1;
      );
      AN    I 102.4;
      AN    M 10.6;
      S     M 10.4;
      A(;
      ON    M 10.2;
      O     M 10.7;
      );
      R     M 10.4;
      NOP   0;
NETWORK
TITLE =
      A     I 91.5;
      AN    I 91.6;
      A     I 91.3;
      AN    I 91.4;
      A(;
      AN    DB100.DBX 110.5;
      A     I 90.1;
      A     I 90.3;
      ON    I 90.1;
      O     DB100.DBX 110.5;
      );
      =     M 10.5;
NETWORK
TITLE =
      A(;
      A     M 10.2;
      A(;
      O     I 102.4;
      O     I 7.0;
      O     I 7.1;
      O     I 7.2;
      );
      S     M 10.6;
      A     M 10.6;
      A(;
      ON    M 10.2;
      O     M 10.7;
      );
      R     M 10.6;
      A     M 10.6;
      );
      A     M 10.5;
      A     DB100.DBX 0.7;
      S     M 10.7;
      A     M 10.7;
      A(;
      O     I 102.3;
      O     DB21.DBX 22.1;
      );
      R     M 10.7;
      NOP   0;
NETWORK
TITLE =
NETWORK
TITLE =
      A     I 7.4;
      BLD   100;
      FP    M 14.1;
      =     M 14.0;
NETWORK
TITLE =
      A     I 7.5;
      BLD   100;
      FP    M 14.3;
      =     M 14.2;
NETWORK
TITLE =
      A     I 7.6;
      BLD   100;
      FP    M 14.5;
      =     M 14.4;
NETWORK
TITLE =
      AN    M 13.1;
      A     I 0.4;
      AN    I 102.3;
      A(;
      O     I 7.0;
      O     M 12.0;
      );
      =     M 12.0;
NETWORK
TITLE =
      AN    M 13.3;
      A     I 0.5;
      AN    I 102.3;
      A(;
      O     I 7.1;
      O     M 12.1;
      );
      =     M 12.1;
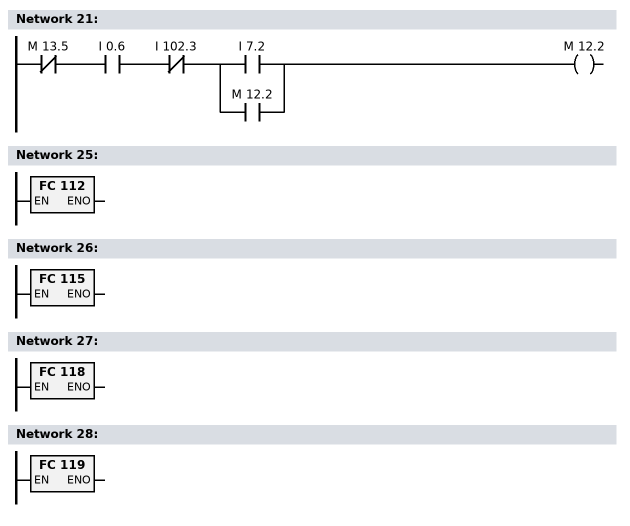
NETWORK
TITLE =
      AN    M 13.5;
      A     I 0.6;
      AN    I 102.3;
      A(;
      O     I 7.2;
      O     M 12.2;
      );
      =     M 12.2;
NETWORK
TITLE =
      A(;
      A(;
      O     M 10.7;
      ON    M 10.4;
      ON    M 10.2;
      );
      AN    Q 3.3;
      A     M 14.0;
      A     M 12.0;
      A(;
      O     M 10.5;
      O     M 1.1;
      );
      AN    M 13.1;
      S     M 13.0;
      A     M 13.0;
      A     M 13.1;
      A     M 14.0;
      A     I 0.4;
      R     M 13.0;
      A     M 13.0;
      );
      S     M 13.1;
      AN    M 13.0;
      A     M 13.1;
      A     M 14.0;
      A     I 0.4;
      R     M 13.1;
      NOP   0;
NETWORK
TITLE =
      A(;
      A(;
      O     M 10.7;
      ON    M 10.4;
      ON    M 10.2;
      );
      AN    Q 3.4;
      A     M 14.2;
      A     M 12.1;
      A(;
      O     M 10.5;
      O     M 1.1;
      );
      AN    M 13.3;
      S     M 13.2;
      A     M 13.2;
      A     M 13.3;
      A     M 14.2;
      A     I 0.5;
      R     M 13.2;
      A     M 13.2;
      );
      S     M 13.3;
      AN    M 13.2;
      A     M 13.3;
      A     M 14.2;
      A     I 0.5;
      R     M 13.3;
      NOP   0;
NETWORK
TITLE =
      A(;
      A(;
      O     M 10.7;
      ON    M 10.4;
      ON    M 10.2;
      );
      AN    Q 3.5;
      A     M 14.4;
      A     M 12.2;
      A(;
      O     M 10.5;
      O     M 1.1;
      );
      AN    M 13.5;
      S     M 13.4;
      A     M 13.4;
      A     M 13.5;
      A     M 14.4;
      A     I 0.6;
      R     M 13.4;
      A     M 13.4;
      );
      S     M 13.5;
      AN    M 13.4;
      A     M 13.5;
      A     M 14.4;
      A     I 0.6;
      R     M 13.5;
      NOP   0;
NETWORK
TITLE =
      CALL  FC 112;
      NOP   0;
NETWORK
TITLE =
      CALL  FC 115;
      NOP   0;
NETWORK
TITLE =
      CALL  FC 118;
      NOP   0;
NETWORK
TITLE =
      CALL  FC 119;
      NOP   0;
END_FUNCTION

FUNCTION FC 112 : VOID
VERSION : 0.1
BEGIN
// (block stored without names or comments; labels and parameter names are numbered)
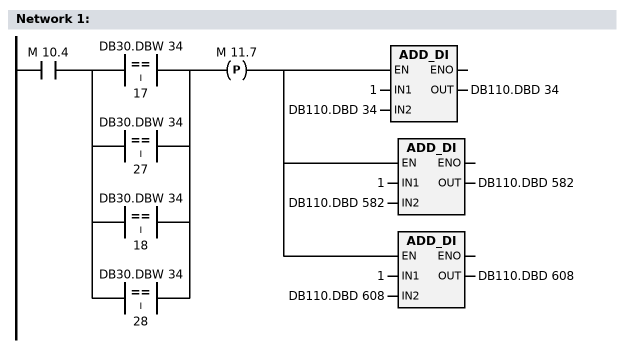
NETWORK
TITLE =
      A     M 10.4;
      A(;
      O(;
      L     DB30.DBW 34;
      L     17;
      ==I;
      );
      O(;
      L     DB30.DBW 34;
      L     27;
      ==I;
      );
      O(;
      L     DB30.DBW 34;
      L     18;
      ==I;
      );
      O(;
      L     DB30.DBW 34;
      L     28;
      ==I;
      );
      );
      FP    M 11.7;
      =     L 0.0;
      A     L 0.0;
      JNB   M001;
      L     1;
      L     DB110.DBD 34;
      +D;
      T     DB110.DBD 34;
M001: NOP   0;
      A     L 0.0;
      JNB   M002;
      L     1;
      L     DB110.DBD 582;
      +D;
      T     DB110.DBD 582;
M002: NOP   0;
      A     L 0.0;
      JNB   M003;
      L     1;
      L     DB110.DBD 608;
      +D;
      T     DB110.DBD 608;
M003: NOP   0;
END_FUNCTION

FUNCTION FC 113 : VOID
VERSION : 0.1
BEGIN
// (block stored without names or comments; labels and parameter names are numbered)
NETWORK
TITLE =
NETWORK
TITLE =
      A(;
      A(;
      A     M 10.4;
      A     M 40.0;
      A     M 40.3;
      A     I 60.0;
      A     I 60.1;
      A(;
      ON    M 120.7;
      O     DB100.DBX 110.1;
      );
      S     M 120.0;
      A(;
      A     M 120.0;
      A     M 120.1;
      ON    M 10.4;
      );
      R     M 120.0;
      A     M 120.0;
      );
      A     DB100.DBX 10.0;
      S     M 120.1;
      A(;
      A     M 120.1;
      A     DB100.DBX 16.1;
      AN    DB100.DBX 10.0;
      ON    M 10.4;
      );
      R     M 120.1;
      A     M 120.1;
      );
      S     DB100.DBX 16.1;
      A     DB100.DBX 16.1;
      A     M 40.3;
      R     DB100.DBX 16.1;
      NOP   0;
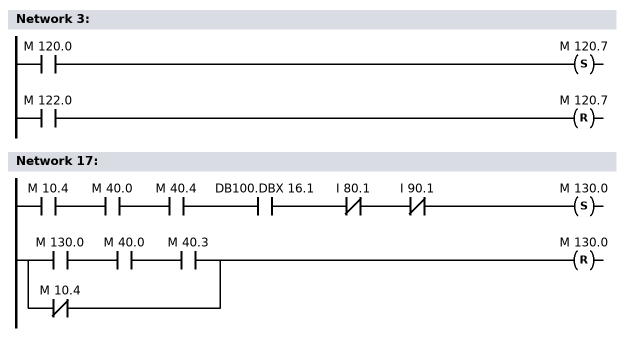
NETWORK
TITLE =
      A     M 120.0;
      S     M 120.7;
      A     M 122.0;
      R     M 120.7;
      NOP   0;
NETWORK
TITLE =
      A(;
      A(;
      A     M 10.4;
      A     M 40.0;
      A     M 40.3;
      AN    I 70.0;
      A     I 70.1;
      A(;
      O     M 120.7;
      O     DB100.DBX 110.0;
      );
      S     M 122.0;
      A(;
      A     M 122.0;
      A     M 122.1;
      ON    M 10.4;
      );
      R     M 122.0;
      A     M 122.0;
      );
      A     DB100.DBX 10.1;
      S     M 122.1;
      A(;
      A     M 122.1;
      A     DB100.DBX 16.1;
      AN    DB100.DBX 10.1;
      ON    M 10.4;
      );
      R     M 122.1;
      A     M 122.1;
      );
      S     DB100.DBX 16.1;
      A     DB100.DBX 16.1;
      A     M 40.3;
      R     DB100.DBX 16.1;
      NOP   0;
NETWORK
TITLE =
NETWORK
TITLE =
      A(;
      A(;
      A     M 10.4;
      A     M 40.0;
      A     M 40.4;
      A     DB100.DBX 16.1;
      A(;
      O     I 80.1;
      O     I 90.1;
      );
      S     M 124.0;
      A(;
      A     M 124.0;
      A     M 124.1;
      ON    M 10.4;
      );
      R     M 124.0;
      A     M 124.0;
      );
      A     DB100.DBX 10.2;
      S     M 124.1;
      A(;
      A     M 124.1;
      A     DB100.DBX 16.5;
      AN    DB100.DBX 10.2;
      ON    M 10.4;
      );
      R     M 124.1;
      A     M 124.1;
      );
      S     DB100.DBX 16.5;
      A     DB100.DBX 16.5;
      A     M 40.3;
      R     DB100.DBX 16.5;
      NOP   0;
NETWORK
TITLE =
NETWORK
TITLE =
      A(;
      A(;
      A     M 10.4;
      A     M 40.1;
      A     M 40.3;
      A(;
      A     DB100.DBX 17.0;
      A(;
      L     DB100.DBW 120;
      L     3;
      ==I;
      );
      O;
      A     DB100.DBX 16.6;
      A(;
      L     DB100.DBW 120;
      L     4;
      ==I;
      );
      );
      S     M 125.0;
      A(;
      A     M 125.0;
      A     M 125.1;
      ON    M 10.4;
      );
      R     M 125.0;
      A     M 125.0;
      );
      A     DB100.DBX 10.3;
      S     M 125.1;
      A(;
      A     M 125.1;
      A     DB100.DBX 16.2;
      AN    DB100.DBX 10.3;
      ON    M 10.4;
      );
      R     M 125.1;
      A     M 125.1;
      );
      A     M 40.1;
      S     DB100.DBX 16.2;
      A     DB100.DBX 16.2;
      A     M 40.0;
      R     DB100.DBX 16.2;
      NOP   0;
NETWORK
TITLE =
      A(;
      A(;
      A     M 10.4;
      A     M 40.0;
      A     M 40.4;
      A(;
      A     DB100.DBX 16.7;
      A(;
      L     DB100.DBW 120;
      L     1;
      ==I;
      );
      O;
      A     DB100.DBX 17.1;
      A(;
      L     DB100.DBW 120;
      L     2;
      ==I;
      );
      );
      S     M 125.2;
      A(;
      A     M 125.0;
      A     M 125.1;
      ON    M 10.4;
      );
      R     M 125.2;
      A     M 125.2;
      );
      A     DB100.DBX 10.3;
      S     M 125.3;
      A(;
      A     M 125.1;
      A     DB100.DBX 16.3;
      AN    DB100.DBX 10.3;
      ON    M 10.4;
      );
      R     M 125.3;
      A     M 125.3;
      );
      A     M 40.4;
      S     DB100.DBX 16.3;
      A     DB100.DBX 16.3;
      A     M 40.3;
      R     DB100.DBX 16.3;
      NOP   0;
NETWORK
TITLE =
NETWORK
TITLE =
      A(;
      A(;
      A     M 10.4;
      A     M 92.6;
      A     M 40.1;
      A     M 40.3;
      A     DB100.DBX 16.6;
      A(;
      L     DB100.DBW 120;
      L     2;
      ==I;
      );
      S     M 126.0;
      A(;
      A     M 126.0;
      A     M 126.1;
      ON    M 10.4;
      );
      R     M 126.0;
      A     M 126.0;
      );
      A     DB100.DBX 10.5;
      S     M 126.1;
      A(;
      A     M 126.1;
      A     DB100.DBX 17.1;
      AN    DB100.DBX 10.5;
      ON    M 10.4;
      );
      R     M 126.1;
      A     M 126.1;
      );
      A     M 40.0;
      A     M 40.4;
      S     DB100.DBX 17.1;
      A     DB100.DBX 17.1;
      A     M 40.3;
      R     DB100.DBX 17.1;
      NOP   0;
NETWORK
TITLE =
      A(;
      A(;
      A     M 10.4;
      A     M 92.6;
      A     M 40.0;
      A     M 40.4;
      A     DB100.DBX 16.5;
      A(;
      O(;
      L     DB100.DBW 120;
      L     1;
      ==I;
      );
      O(;
      L     DB100.DBW 120;
      L     3;
      ==I;
      );
      );
      S     M 126.2;
      A(;
      A     M 126.2;
      A     M 126.3;
      ON    M 10.4;
      );
      R     M 126.2;
      A     M 126.2;
      );
      A     DB100.DBX 10.5;
      S     M 126.3;
      A(;
      A     M 126.3;
      A     DB100.DBX 17.0;
      AN    DB100.DBX 10.5;
      ON    M 10.4;
      );
      R     M 126.3;
      A     M 126.3;
      );
      A     M 40.1;
      A     M 40.3;
      S     DB100.DBX 17.0;
      A     DB100.DBX 17.0;
      A     M 40.0;
      R     DB100.DBX 17.0;
      NOP   0;
NETWORK
TITLE =
NETWORK
TITLE =
      A(;
      A(;
      A     M 10.4;
      A     I 80.0;
      A     I 80.1;
      A     I 80.3;
      A     M 40.1;
      A     M 40.3;
      A     DB100.DBX 17.0;
      A(;
      L     DB100.DBW 120;
      L     1;
      ==I;
      );
      S     M 128.0;
      A(;
      A     M 128.0;
      A     M 128.1;
      ON    M 10.4;
      );
      R     M 128.0;
      A     M 128.0;
      );
      A     DB100.DBX 10.4;
      S     M 128.1;
      A(;
      A     M 128.1;
      A     DB100.DBX 16.7;
      AN    DB100.DBX 10.4;
      ON    M 10.4;
      );
      R     M 128.1;
      A     M 128.1;
      );
      A     M 40.0;
      A     M 40.4;
      S     DB100.DBX 16.7;
      A     DB100.DBX 16.7;
      A     M 40.3;
      R     DB100.DBX 16.7;
      NOP   0;
NETWORK
TITLE =
      A(;
      A(;
      A     M 10.4;
      A     I 80.2;
      A     M 40.0;
      A     M 40.4;
      A     DB100.DBX 16.5;
      A(;
      O(;
      L     DB100.DBW 120;
      L     2;
      ==I;
      );
      O(;
      L     DB100.DBW 120;
      L     4;
      ==I;
      );
      );
      S     M 128.2;
      A(;
      A     M 128.2;
      A     M 128.3;
      ON    M 10.4;
      );
      R     M 128.2;
      A     M 128.2;
      );
      A     DB100.DBX 10.4;
      S     M 128.3;
      A(;
      A     M 128.3;
      A     DB100.DBX 16.6;
      AN    DB100.DBX 10.4;
      ON    M 10.4;
      );
      R     M 128.3;
      A     M 128.3;
      );
      A     M 40.1;
      A     M 40.3;
      S     DB100.DBX 16.6;
      A     DB100.DBX 16.6;
      A     M 40.0;
      R     DB100.DBX 16.6;
      NOP   0;
NETWORK
TITLE =
NETWORK
TITLE =
      A     M 10.4;
      A     M 40.0;
      A     M 40.4;
      A     DB100.DBX 16.1;
      AN    I 80.1;
      AN    I 90.1;
      S     M 130.0;
      A(;
      A     M 130.0;
      A     M 40.0;
      A     M 40.3;
      ON    M 10.4;
      );
      R     M 130.0;
      NOP   0;
END_FUNCTION

FUNCTION FC 115 : VOID
VERSION : 0.1
BEGIN
// (block stored without names or comments; labels and parameter names are numbered)
NETWORK
TITLE =
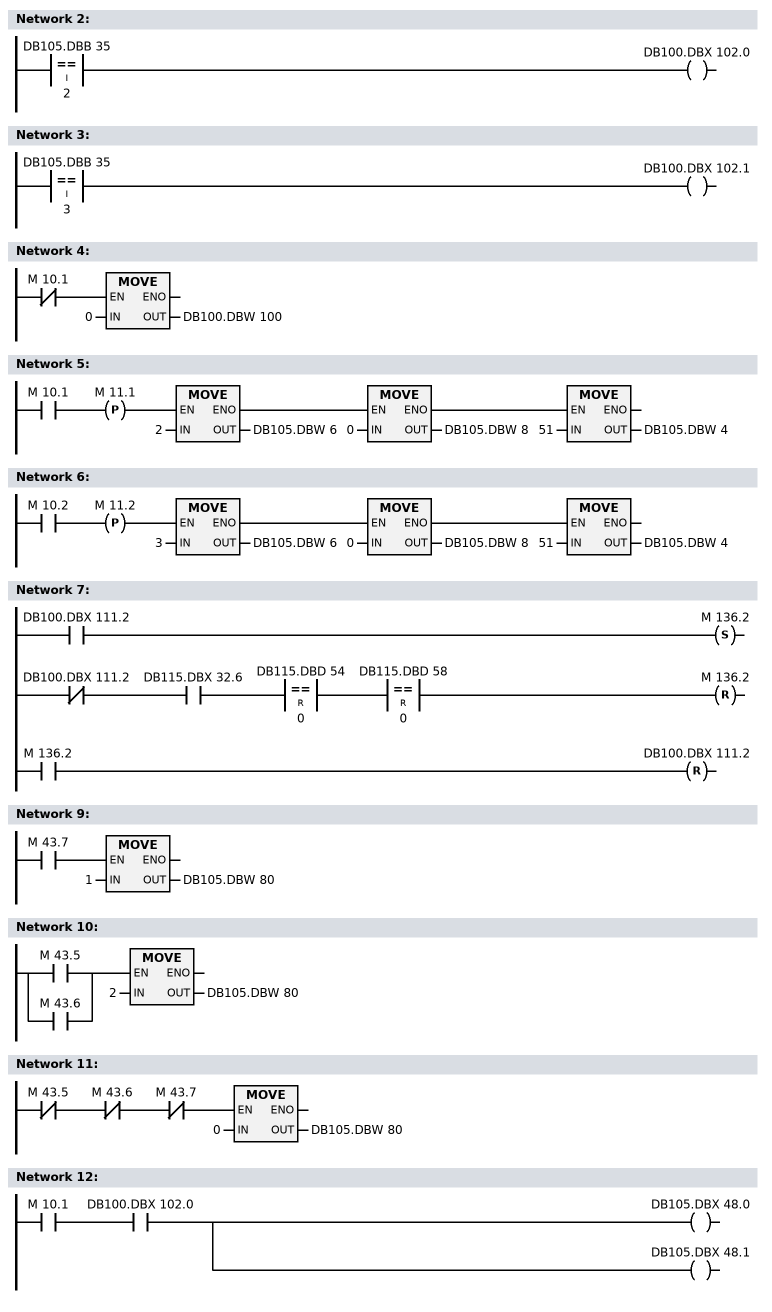
NETWORK
TITLE =
      L     DB105.DBB 35;
      L     2;
      ==I;
      =     DB100.DBX 102.0;
NETWORK
TITLE =
      L     DB105.DBB 35;
      L     3;
      ==I;
      =     DB100.DBX 102.1;
NETWORK
TITLE =
      AN    M 10.1;
      JNB   M001;
      L     0;
      T     DB100.DBW 100;
M001: NOP   0;
NETWORK
TITLE =
      A(;
      A(;
      A     M 10.1;
      FP    M 11.1;
      JNB   M002;
      L     2;
      T     DB105.DBW 6;
      SET;
      SAVE;
      CLR;
M002: A     BR;
      );
      JNB   M003;
      L     0;
      T     DB105.DBW 8;
      SET;
      SAVE;
      CLR;
M003: A     BR;
      );
      JNB   M004;
      L     51;
      T     DB105.DBW 4;
M004: NOP   0;
NETWORK
TITLE =
      A(;
      A(;
      A     M 10.2;
      FP    M 11.2;
      JNB   M005;
      L     3;
      T     DB105.DBW 6;
      SET;
      SAVE;
      CLR;
M005: A     BR;
      );
      JNB   M006;
      L     0;
      T     DB105.DBW 8;
      SET;
      SAVE;
      CLR;
M006: A     BR;
      );
      JNB   M007;
      L     51;
      T     DB105.DBW 4;
M007: NOP   0;
NETWORK
TITLE =
      A     DB100.DBX 111.2;
      S     M 136.2;
      AN    DB100.DBX 111.2;
      A     DB115.DBX 32.6;
      A(;
      L     DB115.DBD 54;
      L     0;
      ==R;
      );
      A(;
      L     DB115.DBD 58;
      L     0;
      ==R;
      );
      R     M 136.2;
      A     M 136.2;
      R     DB100.DBX 111.2;
NETWORK
TITLE =
NETWORK
TITLE =
      A     M 43.7;
      JNB   M008;
      L     1;
      T     DB105.DBW 80;
M008: NOP   0;
NETWORK
TITLE =
      A(;
      O     M 43.5;
      O     M 43.6;
      );
      JNB   M009;
      L     2;
      T     DB105.DBW 80;
M009: NOP   0;
NETWORK
TITLE =
      AN    M 43.5;
      AN    M 43.6;
      AN    M 43.7;
      JNB   M010;
      L     0;
      T     DB105.DBW 80;
M010: NOP   0;
NETWORK
TITLE =
      A     M 10.1;
      A     DB100.DBX 102.0;
      =     DB105.DBX 48.0;
      =     DB105.DBX 48.1;
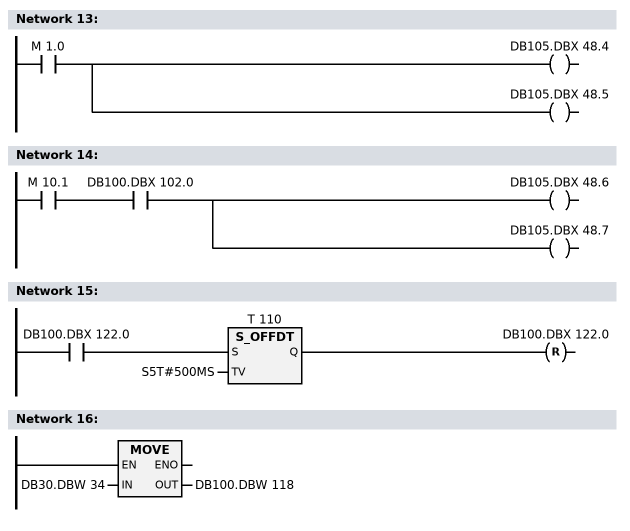
NETWORK
TITLE =
      A     M 1.0;
      =     DB105.DBX 48.4;
      =     DB105.DBX 48.5;
NETWORK
TITLE =
      A     M 10.1;
      A     DB100.DBX 102.0;
      =     DB105.DBX 48.6;
      =     DB105.DBX 48.7;
NETWORK
TITLE =
      A     DB100.DBX 122.0;
      L     S5T#500MS;
      SF    T 110;
      NOP   0;
      NOP   0;
      NOP   0;
      A     T 110;
      R     DB100.DBX 122.0;
NETWORK
TITLE =
      L     DB30.DBW 34;
      T     DB100.DBW 118;
      NOP   0;
END_FUNCTION

FUNCTION FC 118 : VOID
VERSION : 0.1
BEGIN
// (block stored without names or comments; labels and parameter names are numbered)
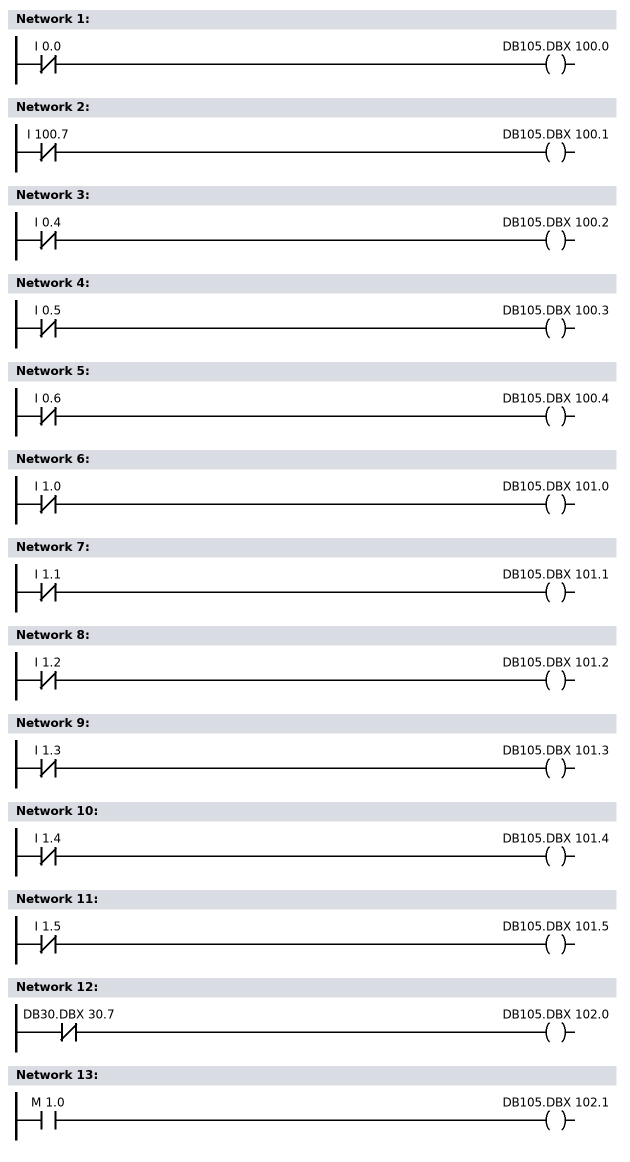
NETWORK
TITLE =
      AN    I 0.0;
      =     DB105.DBX 100.0;
NETWORK
TITLE =
      AN    I 100.7;
      =     DB105.DBX 100.1;
NETWORK
TITLE =
      AN    I 0.4;
      =     DB105.DBX 100.2;
NETWORK
TITLE =
      AN    I 0.5;
      =     DB105.DBX 100.3;
NETWORK
TITLE =
      AN    I 0.6;
      =     DB105.DBX 100.4;
NETWORK
TITLE =
      AN    I 1.0;
      =     DB105.DBX 101.0;
NETWORK
TITLE =
      AN    I 1.1;
      =     DB105.DBX 101.1;
NETWORK
TITLE =
      AN    I 1.2;
      =     DB105.DBX 101.2;
NETWORK
TITLE =
      AN    I 1.3;
      =     DB105.DBX 101.3;
NETWORK
TITLE =
      AN    I 1.4;
      =     DB105.DBX 101.4;
NETWORK
TITLE =
      AN    I 1.5;
      =     DB105.DBX 101.5;
NETWORK
TITLE =
      AN    DB30.DBX 30.7;
      =     DB105.DBX 102.0;
NETWORK
TITLE =
      A     M 1.0;
      =     DB105.DBX 102.1;
NETWORK
TITLE =
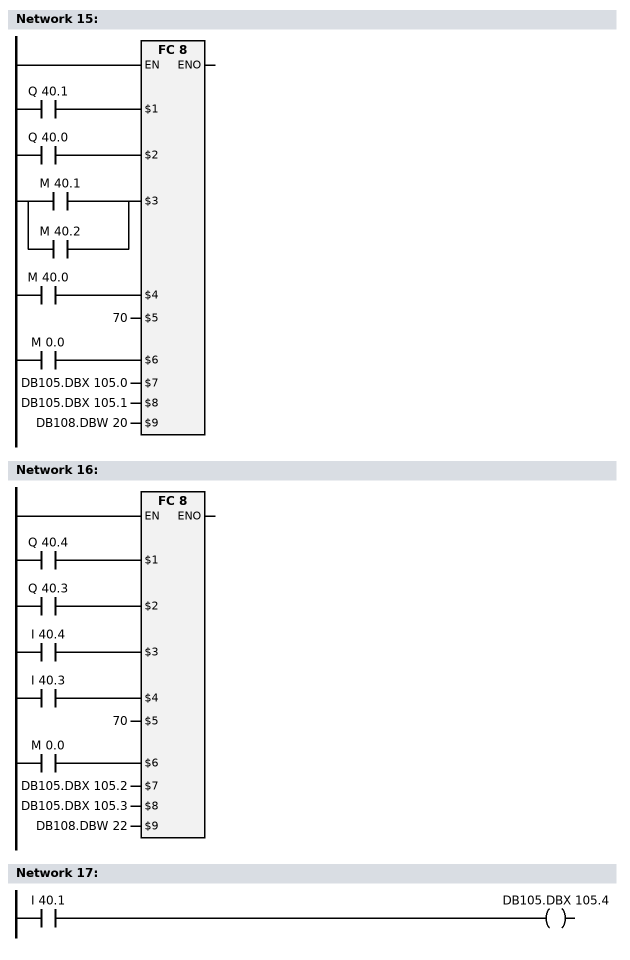
NETWORK
TITLE =
      A     Q 40.1;
      =     L 0.0;
      BLD   103;
      A     Q 40.0;
      =     L 0.1;
      BLD   103;
      A(;
      O     M 40.1;
      O     M 40.2;
      );
      =     L 0.2;
      BLD   103;
      A     M 40.0;
      =     L 0.3;
      BLD   103;
      A     M 0.0;
      =     L 0.4;
      BLD   103;
      CALL  FC 8 (
           $1                       := L 0.0,
           $2                       := L 0.1,
           $3                       := L 0.2,
           $4                       := L 0.3,
           $5                       := 70,
           $6                       := L 0.4,
           $7                       := DB105.DBX 105.0,
           $8                       := DB105.DBX 105.1,
           $9                       := DB108.DBW 20);
      NOP   0;
NETWORK
TITLE =
      A     Q 40.4;
      =     L 0.0;
      BLD   103;
      A     Q 40.3;
      =     L 0.1;
      BLD   103;
      A     I 40.4;
      =     L 0.2;
      BLD   103;
      A     I 40.3;
      =     L 0.3;
      BLD   103;
      A     M 0.0;
      =     L 0.4;
      BLD   103;
      CALL  FC 8 (
           $1                       := L 0.0,
           $2                       := L 0.1,
           $3                       := L 0.2,
           $4                       := L 0.3,
           $5                       := 70,
           $6                       := L 0.4,
           $7                       := DB105.DBX 105.2,
           $8                       := DB105.DBX 105.3,
           $9                       := DB108.DBW 22);
      NOP   0;
NETWORK
TITLE =
      A     I 40.1;
      =     DB105.DBX 105.4;
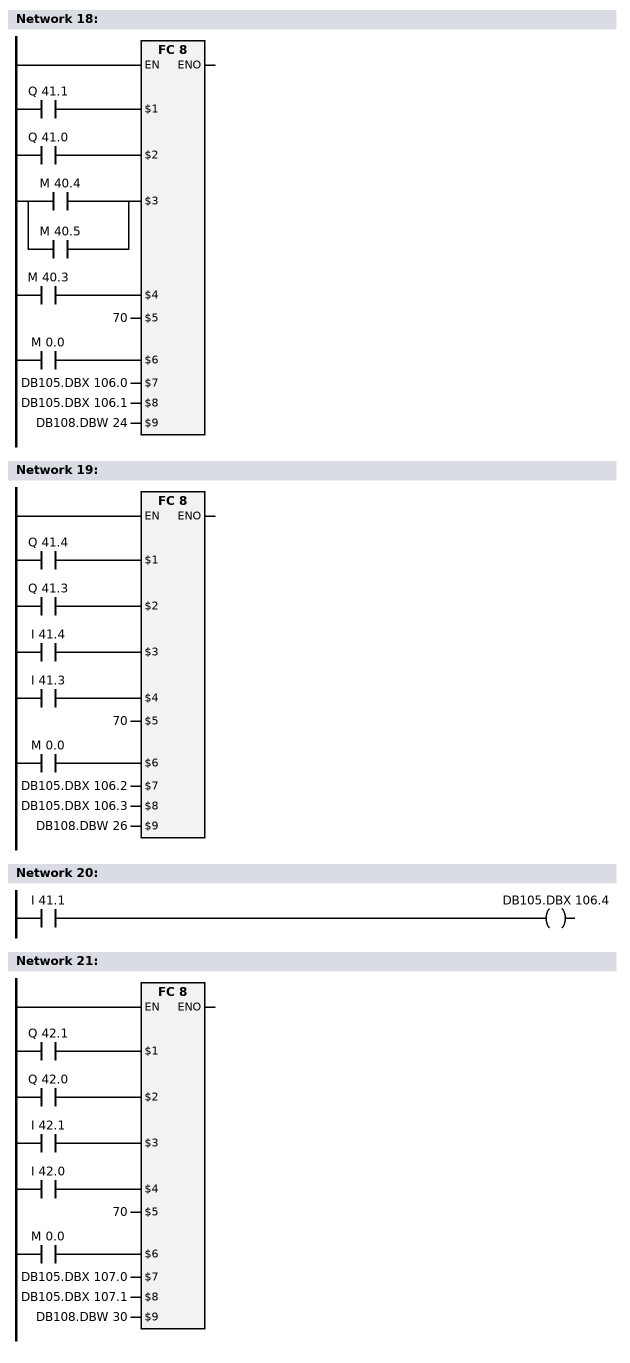
NETWORK
TITLE =
      A     Q 41.1;
      =     L 0.0;
      BLD   103;
      A     Q 41.0;
      =     L 0.1;
      BLD   103;
      A(;
      O     M 40.4;
      O     M 40.5;
      );
      =     L 0.2;
      BLD   103;
      A     M 40.3;
      =     L 0.3;
      BLD   103;
      A     M 0.0;
      =     L 0.4;
      BLD   103;
      CALL  FC 8 (
           $1                       := L 0.0,
           $2                       := L 0.1,
           $3                       := L 0.2,
           $4                       := L 0.3,
           $5                       := 70,
           $6                       := L 0.4,
           $7                       := DB105.DBX 106.0,
           $8                       := DB105.DBX 106.1,
           $9                       := DB108.DBW 24);
      NOP   0;
NETWORK
TITLE =
      A     Q 41.4;
      =     L 0.0;
      BLD   103;
      A     Q 41.3;
      =     L 0.1;
      BLD   103;
      A     I 41.4;
      =     L 0.2;
      BLD   103;
      A     I 41.3;
      =     L 0.3;
      BLD   103;
      A     M 0.0;
      =     L 0.4;
      BLD   103;
      CALL  FC 8 (
           $1                       := L 0.0,
           $2                       := L 0.1,
           $3                       := L 0.2,
           $4                       := L 0.3,
           $5                       := 70,
           $6                       := L 0.4,
           $7                       := DB105.DBX 106.2,
           $8                       := DB105.DBX 106.3,
           $9                       := DB108.DBW 26);
      NOP   0;
NETWORK
TITLE =
      A     I 41.1;
      =     DB105.DBX 106.4;
NETWORK
TITLE =
      A     Q 42.1;
      =     L 0.0;
      BLD   103;
      A     Q 42.0;
      =     L 0.1;
      BLD   103;
      A     I 42.1;
      =     L 0.2;
      BLD   103;
      A     I 42.0;
      =     L 0.3;
      BLD   103;
      A     M 0.0;
      =     L 0.4;
      BLD   103;
      CALL  FC 8 (
           $1                       := L 0.0,
           $2                       := L 0.1,
           $3                       := L 0.2,
           $4                       := L 0.3,
           $5                       := 70,
           $6                       := L 0.4,
           $7                       := DB105.DBX 107.0,
           $8                       := DB105.DBX 107.1,
           $9                       := DB108.DBW 30);
      NOP   0;
NETWORK
TITLE =
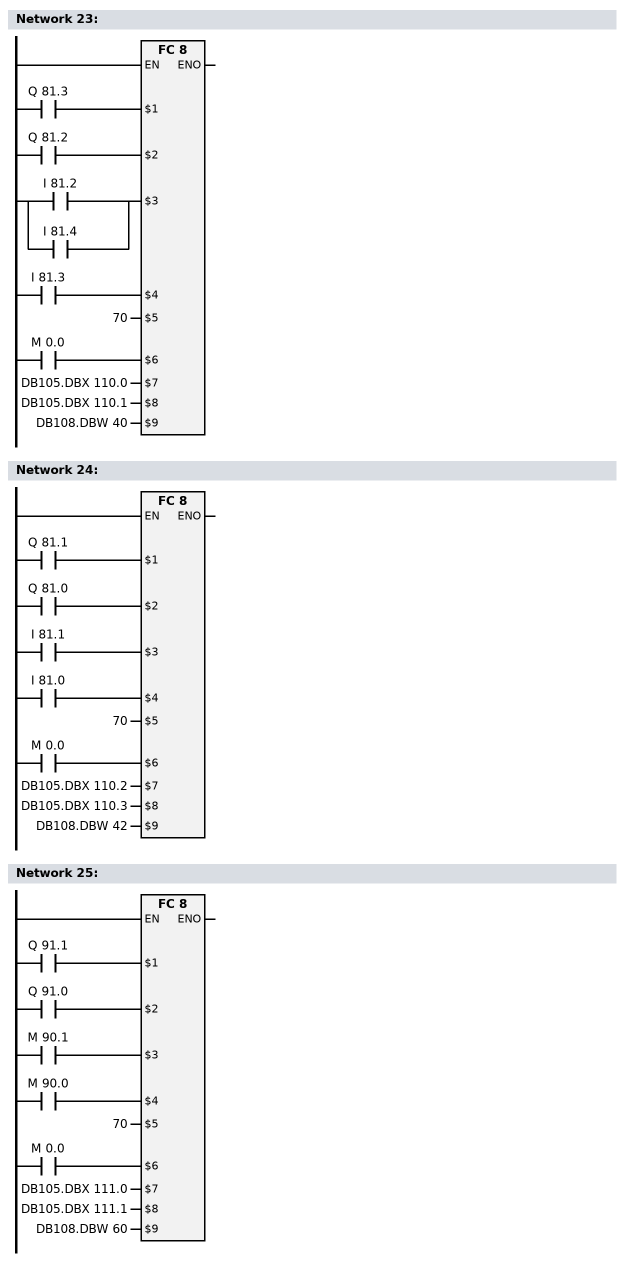
NETWORK
TITLE =
      A     Q 81.3;
      =     L 0.0;
      BLD   103;
      A     Q 81.2;
      =     L 0.1;
      BLD   103;
      A(;
      O     I 81.2;
      O     I 81.4;
      );
      =     L 0.2;
      BLD   103;
      A     I 81.3;
      =     L 0.3;
      BLD   103;
      A     M 0.0;
      =     L 0.4;
      BLD   103;
      CALL  FC 8 (
           $1                       := L 0.0,
           $2                       := L 0.1,
           $3                       := L 0.2,
           $4                       := L 0.3,
           $5                       := 70,
           $6                       := L 0.4,
           $7                       := DB105.DBX 110.0,
           $8                       := DB105.DBX 110.1,
           $9                       := DB108.DBW 40);
      NOP   0;
NETWORK
TITLE =
      A     Q 81.1;
      =     L 0.0;
      BLD   103;
      A     Q 81.0;
      =     L 0.1;
      BLD   103;
      A     I 81.1;
      =     L 0.2;
      BLD   103;
      A     I 81.0;
      =     L 0.3;
      BLD   103;
      A     M 0.0;
      =     L 0.4;
      BLD   103;
      CALL  FC 8 (
           $1                       := L 0.0,
           $2                       := L 0.1,
           $3                       := L 0.2,
           $4                       := L 0.3,
           $5                       := 70,
           $6                       := L 0.4,
           $7                       := DB105.DBX 110.2,
           $8                       := DB105.DBX 110.3,
           $9                       := DB108.DBW 42);
      NOP   0;
NETWORK
TITLE =
      A     Q 91.1;
      =     L 0.0;
      BLD   103;
      A     Q 91.0;
      =     L 0.1;
      BLD   103;
      A     M 90.1;
      =     L 0.2;
      BLD   103;
      A     M 90.0;
      =     L 0.3;
      BLD   103;
      A     M 0.0;
      =     L 0.4;
      BLD   103;
      CALL  FC 8 (
           $1                       := L 0.0,
           $2                       := L 0.1,
           $3                       := L 0.2,
           $4                       := L 0.3,
           $5                       := 70,
           $6                       := L 0.4,
           $7                       := DB105.DBX 111.0,
           $8                       := DB105.DBX 111.1,
           $9                       := DB108.DBW 60);
      NOP   0;
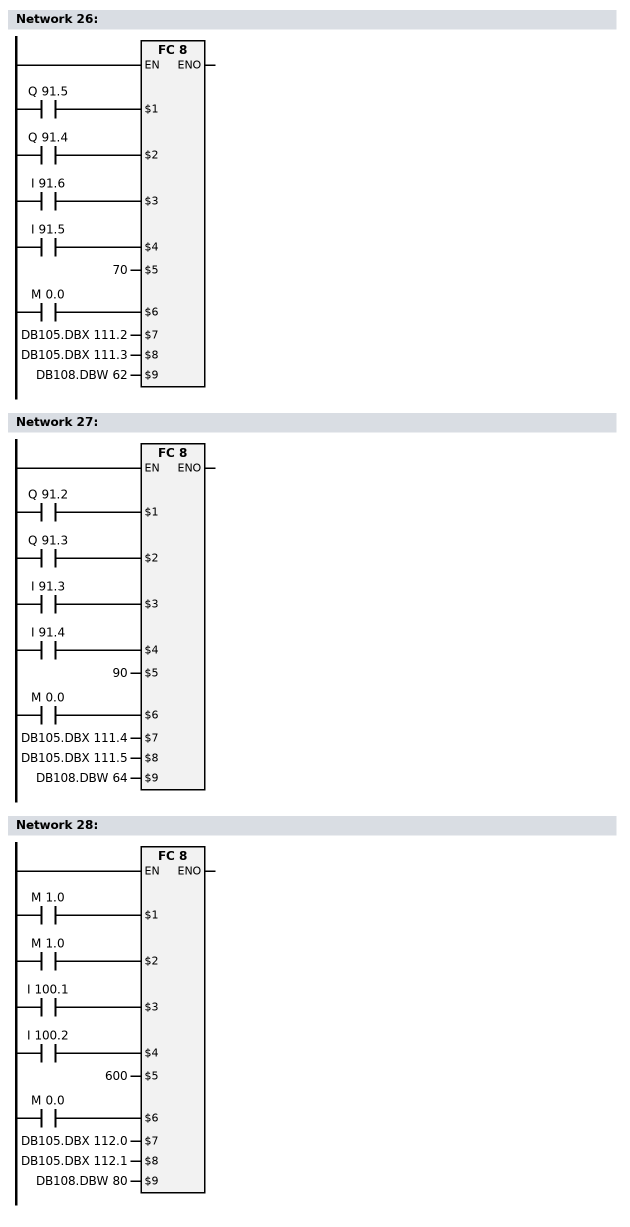
NETWORK
TITLE =
      A     Q 91.5;
      =     L 0.0;
      BLD   103;
      A     Q 91.4;
      =     L 0.1;
      BLD   103;
      A     I 91.6;
      =     L 0.2;
      BLD   103;
      A     I 91.5;
      =     L 0.3;
      BLD   103;
      A     M 0.0;
      =     L 0.4;
      BLD   103;
      CALL  FC 8 (
           $1                       := L 0.0,
           $2                       := L 0.1,
           $3                       := L 0.2,
           $4                       := L 0.3,
           $5                       := 70,
           $6                       := L 0.4,
           $7                       := DB105.DBX 111.2,
           $8                       := DB105.DBX 111.3,
           $9                       := DB108.DBW 62);
      NOP   0;
NETWORK
TITLE =
      A     Q 91.2;
      =     L 0.0;
      BLD   103;
      A     Q 91.3;
      =     L 0.1;
      BLD   103;
      A     I 91.3;
      =     L 0.2;
      BLD   103;
      A     I 91.4;
      =     L 0.3;
      BLD   103;
      A     M 0.0;
      =     L 0.4;
      BLD   103;
      CALL  FC 8 (
           $1                       := L 0.0,
           $2                       := L 0.1,
           $3                       := L 0.2,
           $4                       := L 0.3,
           $5                       := 90,
           $6                       := L 0.4,
           $7                       := DB105.DBX 111.4,
           $8                       := DB105.DBX 111.5,
           $9                       := DB108.DBW 64);
      NOP   0;
NETWORK
TITLE =
      A     M 1.0;
      =     L 0.0;
      BLD   103;
      A     M 1.0;
      =     L 0.1;
      BLD   103;
      A     I 100.1;
      =     L 0.2;
      BLD   103;
      A     I 100.2;
      =     L 0.3;
      BLD   103;
      A     M 0.0;
      =     L 0.4;
      BLD   103;
      CALL  FC 8 (
           $1                       := L 0.0,
           $2                       := L 0.1,
           $3                       := L 0.2,
           $4                       := L 0.3,
           $5                       := 600,
           $6                       := L 0.4,
           $7                       := DB105.DBX 112.0,
           $8                       := DB105.DBX 112.1,
           $9                       := DB108.DBW 80);
      NOP   0;
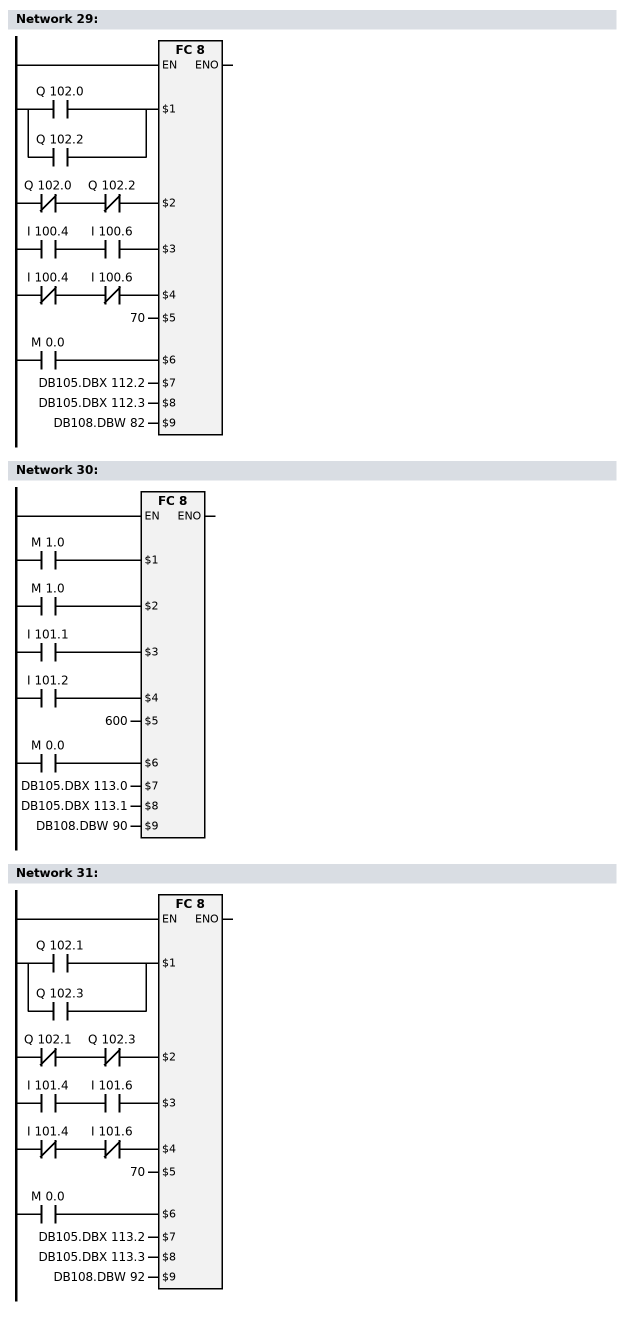
NETWORK
TITLE =
      A(;
      O     Q 102.0;
      O     Q 102.2;
      );
      =     L 0.0;
      BLD   103;
      AN    Q 102.0;
      AN    Q 102.2;
      =     L 0.1;
      BLD   103;
      A     I 100.4;
      A     I 100.6;
      =     L 0.2;
      BLD   103;
      AN    I 100.4;
      AN    I 100.6;
      =     L 0.3;
      BLD   103;
      A     M 0.0;
      =     L 0.4;
      BLD   103;
      CALL  FC 8 (
           $1                       := L 0.0,
           $2                       := L 0.1,
           $3                       := L 0.2,
           $4                       := L 0.3,
           $5                       := 70,
           $6                       := L 0.4,
           $7                       := DB105.DBX 112.2,
           $8                       := DB105.DBX 112.3,
           $9                       := DB108.DBW 82);
      NOP   0;
NETWORK
TITLE =
      A     M 1.0;
      =     L 0.0;
      BLD   103;
      A     M 1.0;
      =     L 0.1;
      BLD   103;
      A     I 101.1;
      =     L 0.2;
      BLD   103;
      A     I 101.2;
      =     L 0.3;
      BLD   103;
      A     M 0.0;
      =     L 0.4;
      BLD   103;
      CALL  FC 8 (
           $1                       := L 0.0,
           $2                       := L 0.1,
           $3                       := L 0.2,
           $4                       := L 0.3,
           $5                       := 600,
           $6                       := L 0.4,
           $7                       := DB105.DBX 113.0,
           $8                       := DB105.DBX 113.1,
           $9                       := DB108.DBW 90);
      NOP   0;
NETWORK
TITLE =
      A(;
      O     Q 102.1;
      O     Q 102.3;
      );
      =     L 0.0;
      BLD   103;
      AN    Q 102.1;
      AN    Q 102.3;
      =     L 0.1;
      BLD   103;
      A     I 101.4;
      A     I 101.6;
      =     L 0.2;
      BLD   103;
      AN    I 101.4;
      AN    I 101.6;
      =     L 0.3;
      BLD   103;
      A     M 0.0;
      =     L 0.4;
      BLD   103;
      CALL  FC 8 (
           $1                       := L 0.0,
           $2                       := L 0.1,
           $3                       := L 0.2,
           $4                       := L 0.3,
           $5                       := 70,
           $6                       := L 0.4,
           $7                       := DB105.DBX 113.2,
           $8                       := DB105.DBX 113.3,
           $9                       := DB108.DBW 92);
      NOP   0;
